// TIA Portal V17 program export: 0 tag tables, 0 data types, 33 data blocks, 57 code blocks (in call order from the OBs), 62 instance data blocks

DATA_BLOCK "DB_MainData"   // DB5001
{ S7_Optimized_Access := 'TRUE' }
VERSION : 0.1
// stored: AutoNumber false, DBAccessibleFromOPCUA true, DBAccessibleFromWebserver true, IsOnlyStoredInLoadMemory false, IsRetainMemResEnabled false, IsWriteProtectedInAS false, MemoryReserve 100
   VAR
      SafetyLevels { S7_SetPoint := 'True'} : "UDT_SafetyLevels";
      HMI { S7_SetPoint := 'True'} : "UDT_HMI";
      ManualModeActive : Bool := FALSE;
      MachineMode : UInt := 1;   // 0= No mode active, 1= Manual mode, 2= Homing mode, 3= Automatic mode
      AntennaEdge : Bool := FALSE;
      Antenna : Bool := FALSE;
   END_VAR
BEGIN
   SafetyLevels."Level_1L+" := FALSE;
   SafetyLevels."Level_2L+" := FALSE;
   SafetyLevels."Level_3L+" := TRUE;   // Doors + safety barriers + total stop
   SafetyLevels."Level_4L+" := FALSE;   // Doors + safety barriers + total stop + light barriers
   SafetyLevels."Level_5L+" := FALSE;   // Doors + safety barriers + total stop + turn table
   SafetyLevels."Level_6L+" := FALSE;
   SafetyLevels."Level_7L+" := FALSE;
   SafetyLevels."Level_8L+" := FALSE;
   SafetyLevels."Level_9L+" := FALSE;
   SafetyLevels."Level_10L+" := FALSE;
   SafetyLevels.SystemReady := TRUE;   // Doors + safety barriers + total stop + air pressure
   HMI.ScreenData[1] := 16#0001;
   HMI.ScreenData[2] := 16#0008;
   HMI.ScreenData[3] := 16#0000;
   HMI.ScreenData[4] := 16#0007;
   HMI.ScreenData[5] := 16#0000;
   HMI.UserNumber := 0;
   HMI.ActualScreenNumber := 8;
   HMI.RequiredScreenNumber := 0;
   HMI.FunctionKeys[1..8] := FALSE;
END_DATA_BLOCK

DATA_BLOCK "READER_DWELL"   // DB80
{ S7_Optimized_Access := 'TRUE' }
VERSION : 0.1
// stored: AutoNumber true, DBAccessibleFromOPCUA true, DBAccessibleFromWebserver true, IsOnlyStoredInLoadMemory false, IsRetainMemResEnabled false, IsWriteProtectedInAS false, MemoryReserve 100
   VAR
      DWELL_TMR : Array[0..16] of TON_TIME;
   END_VAR
BEGIN
END_DATA_BLOCK

DATA_BLOCK "Alarms"   // DB20
{ S7_Optimized_Access := 'FALSE' }
VERSION : 0.1
// stored: AutoNumber false, DBAccessibleFromOPCUA true, DBAccessibleFromWebserver true, IsOnlyStoredInLoadMemory false, IsWriteProtectedInAS false
   VAR
      Alarm : Array[1..256] of Bool;
      Warning : Array[1..256] of Bool;
      PartErrorsHMI : Array[1..256] of Bool;
      NOKInAuto : Bool := FALSE;
      Reset : Bool := FALSE;
      ResetHmi : Bool := FALSE;
      AlarmPLC : Array[0..100] of Bool;
   END_VAR
BEGIN
   Alarm[1..256] := FALSE;
   Warning[1..256] := FALSE;
   PartErrorsHMI[1..10] := FALSE;
   PartErrorsHMI[11] := TRUE;
   PartErrorsHMI[12..20] := FALSE;
   PartErrorsHMI[21] := TRUE;
   PartErrorsHMI[22..30] := FALSE;
   PartErrorsHMI[31] := TRUE;
   PartErrorsHMI[32..40] := FALSE;
   PartErrorsHMI[41] := TRUE;
   PartErrorsHMI[42..256] := FALSE;
   AlarmPLC[0..100] := FALSE;
END_DATA_BLOCK

DATA_BLOCK "AutoInfo"   // DB13
{ S7_Optimized_Access := 'TRUE' }
VERSION : 0.1
// stored: AutoNumber true, DBAccessibleFromOPCUA true, DBAccessibleFromWebserver true, IsOnlyStoredInLoadMemory false, IsRetainMemResEnabled false, IsWriteProtectedInAS false, MemoryReserve 100
   VAR
      EraseStation : Array[1..8] of Bool;
      ExtractedScan : String := '';
      EnableReferenceChange : Bool := TRUE;
   END_VAR
   VAR RETAIN
      R1BrakeTestRequired : Bool := TRUE;
      R1MasteringRequired : Bool := TRUE;
      PartMeasuredData { S7_SetPoint := 'True'} : "UDT_MeasuredPartData";
   END_VAR
   VAR
      EndProduction { S7_SetPoint := 'True'} : Bool;
   END_VAR
BEGIN
   EraseStation[1..8] := FALSE;
   PartMeasuredData.LeftCupforming.MaxForce := -7.98946;
   PartMeasuredData.LeftCupforming.MinimalWay := 9.841429;
   PartMeasuredData.LeftCupforming.MaxZposition := 55.44488;
   PartMeasuredData.LeftCupforming.OK := TRUE;
   PartMeasuredData.LeftCupforming.NOK := FALSE;
   PartMeasuredData.LeftCupforming.parameters.DigiforceProgram := 1;
   PartMeasuredData.LeftCupforming.parameters.FinalSpeed := 20.0;
   PartMeasuredData.LeftCupforming.parameters.ApproachSpeed := 100.0;
   PartMeasuredData.LeftCupforming.parameters.FinalForce := 80.0;
   PartMeasuredData.LeftCupforming.parameters.ApproachForce := 20.0;
   PartMeasuredData.LeftCupforming.parameters.EndWayImmediate := 9.9;
   PartMeasuredData.LeftCupforming.parameters.EndWayWithTimeout := 9.9;
   PartMeasuredData.LeftCupforming.parameters.SwitchingWay := 50.0;
   PartMeasuredData.LeftCupforming.parameters.EndWayTimeout := T#300MS;
   PartMeasuredData.RightCupforming.MaxForce := 8.163286;
   PartMeasuredData.RightCupforming.MinimalWay := 9.87697;
   PartMeasuredData.RightCupforming.MaxZposition := 56.52127;
   PartMeasuredData.RightCupforming.OK := TRUE;
   PartMeasuredData.RightCupforming.NOK := FALSE;
   PartMeasuredData.RightCupforming.parameters.DigiforceProgram := 1;
   PartMeasuredData.RightCupforming.parameters.FinalSpeed := 20.0;
   PartMeasuredData.RightCupforming.parameters.ApproachSpeed := 100.0;
   PartMeasuredData.RightCupforming.parameters.FinalForce := 80.0;
   PartMeasuredData.RightCupforming.parameters.ApproachForce := 20.0;
   PartMeasuredData.RightCupforming.parameters.EndWayImmediate := 9.9;
   PartMeasuredData.RightCupforming.parameters.EndWayWithTimeout := 9.9;
   PartMeasuredData.RightCupforming.parameters.SwitchingWay := 50.0;
   PartMeasuredData.RightCupforming.parameters.EndWayTimeout := T#300MS;
   PartMeasuredData.LeftRiveting1.Start := FALSE;
   PartMeasuredData.LeftRiveting1.PrgNumber := 0;
   PartMeasuredData.LeftRiveting1.Ready := FALSE;
   PartMeasuredData.LeftRiveting1.Running := FALSE;
   PartMeasuredData.LeftRiveting1.OK := FALSE;
   PartMeasuredData.LeftRiveting1.NOK := FALSE;
   PartMeasuredData.LeftRiveting1.H1OK := FALSE;
   PartMeasuredData.LeftRiveting1.H2OK := FALSE;
   PartMeasuredData.LeftRiveting1.TimeOK := FALSE;
   PartMeasuredData.LeftRiveting1.StartError := FALSE;
   PartMeasuredData.LeftRiveting1.LastH1 := 0.0;
   PartMeasuredData.LeftRiveting1.LastH2 := 0.0;
   PartMeasuredData.LeftRiveting1.LastTime := 0.0;
   PartMeasuredData.LeftRiveting1.LastZ1 := 0.0;
   PartMeasuredData.LeftRiveting1.Error := FALSE;
   PartMeasuredData.LeftRiveting1.NewData := FALSE;
   PartMeasuredData.LeftRiveting1.Z1OK := FALSE;
   PartMeasuredData.LeftRiveting1.NewDataAfterStart := FALSE;
   PartMeasuredData.LeftRiveting1.LastZ2 := 0.0;
   PartMeasuredData.LeftRiveting2.Start := FALSE;
   PartMeasuredData.LeftRiveting2.PrgNumber := 0;
   PartMeasuredData.LeftRiveting2.Ready := FALSE;
   PartMeasuredData.LeftRiveting2.Running := FALSE;
   PartMeasuredData.LeftRiveting2.OK := FALSE;
   PartMeasuredData.LeftRiveting2.NOK := FALSE;
   PartMeasuredData.LeftRiveting2.H1OK := FALSE;
   PartMeasuredData.LeftRiveting2.H2OK := FALSE;
   PartMeasuredData.LeftRiveting2.TimeOK := FALSE;
   PartMeasuredData.LeftRiveting2.StartError := FALSE;
   PartMeasuredData.LeftRiveting2.LastH1 := 0.0;
   PartMeasuredData.LeftRiveting2.LastH2 := 0.0;
   PartMeasuredData.LeftRiveting2.LastTime := 0.0;
   PartMeasuredData.LeftRiveting2.LastZ1 := 0.0;
   PartMeasuredData.LeftRiveting2.Error := FALSE;
   PartMeasuredData.LeftRiveting2.NewData := FALSE;
   PartMeasuredData.LeftRiveting2.Z1OK := FALSE;
   PartMeasuredData.LeftRiveting2.NewDataAfterStart := FALSE;
   PartMeasuredData.LeftRiveting2.LastZ2 := 0.0;
   PartMeasuredData.RightRiveting1.Start := FALSE;
   PartMeasuredData.RightRiveting1.PrgNumber := 0;
   PartMeasuredData.RightRiveting1.Ready := FALSE;
   PartMeasuredData.RightRiveting1.Running := FALSE;
   PartMeasuredData.RightRiveting1.OK := FALSE;
   PartMeasuredData.RightRiveting1.NOK := FALSE;
   PartMeasuredData.RightRiveting1.H1OK := FALSE;
   PartMeasuredData.RightRiveting1.H2OK := FALSE;
   PartMeasuredData.RightRiveting1.TimeOK := FALSE;
   PartMeasuredData.RightRiveting1.StartError := FALSE;
   PartMeasuredData.RightRiveting1.LastH1 := 0.0;
   PartMeasuredData.RightRiveting1.LastH2 := 0.0;
   PartMeasuredData.RightRiveting1.LastTime := 0.0;
   PartMeasuredData.RightRiveting1.LastZ1 := 0.0;
   PartMeasuredData.RightRiveting1.Error := FALSE;
   PartMeasuredData.RightRiveting1.NewData := FALSE;
   PartMeasuredData.RightRiveting1.Z1OK := FALSE;
   PartMeasuredData.RightRiveting1.NewDataAfterStart := FALSE;
   PartMeasuredData.RightRiveting1.LastZ2 := 0.0;
   PartMeasuredData.RightRiveting2.Start := FALSE;
   PartMeasuredData.RightRiveting2.PrgNumber := 0;
   PartMeasuredData.RightRiveting2.Ready := FALSE;
   PartMeasuredData.RightRiveting2.Running := FALSE;
   PartMeasuredData.RightRiveting2.OK := FALSE;
   PartMeasuredData.RightRiveting2.NOK := FALSE;
   PartMeasuredData.RightRiveting2.H1OK := FALSE;
   PartMeasuredData.RightRiveting2.H2OK := FALSE;
   PartMeasuredData.RightRiveting2.TimeOK := FALSE;
   PartMeasuredData.RightRiveting2.StartError := FALSE;
   PartMeasuredData.RightRiveting2.LastH1 := 0.0;
   PartMeasuredData.RightRiveting2.LastH2 := 0.0;
   PartMeasuredData.RightRiveting2.LastTime := 0.0;
   PartMeasuredData.RightRiveting2.LastZ1 := 0.0;
   PartMeasuredData.RightRiveting2.Error := FALSE;
   PartMeasuredData.RightRiveting2.NewData := FALSE;
   PartMeasuredData.RightRiveting2.Z1OK := FALSE;
   PartMeasuredData.RightRiveting2.NewDataAfterStart := FALSE;
   PartMeasuredData.RightRiveting2.LastZ2 := 0.0;
END_DATA_BLOCK

DATA_BLOCK "AutoPositions"   // DB11
{ S7_Optimized_Access := 'TRUE' }
VERSION : 0.1
// stored: AutoNumber true, DBAccessibleFromOPCUA true, DBAccessibleFromWebserver true, IsOnlyStoredInLoadMemory false, IsRetainMemResEnabled false, IsWriteProtectedInAS false, MemoryReserve 100
   VAR RETAIN
      St1_Table1 : "UDT_PositionData";
      St2_Table2 : "UDT_PositionData";
      St3_Fitting : "UDT_PositionData";
      R1_Gripper : "UDT_PositionData";
      AE_Gripper : "UDT_PositionData";
      St4_OKposition : "UDT_PositionData";
   END_VAR
   VAR
      emptyPos : "UDT_PositionData";
   END_VAR
BEGIN
END_DATA_BLOCK

DATA_BLOCK "St1Insertion"   // DB15
{ S7_Optimized_Access := 'TRUE' }
VERSION : 0.1
// stored: AutoNumber true, DBAccessibleFromOPCUA true, DBAccessibleFromWebserver true, IsOnlyStoredInLoadMemory false, IsRetainMemResEnabled false, IsWriteProtectedInAS false, MemoryReserve 100
   VAR
      ExpectedSensors : Array[0..20] of Bool;
      UsedSensors : Array[0..20] of Bool;
      SensorsState : Array[0..20] of Bool;
      SensorsNOK : Array[0..20] of Bool;
      NOKList : Array[0..20] of Int;
      InsertionOK : Bool := TRUE;
      InsertionNOK : Bool := FALSE;
      InsertionEmpty : Bool := TRUE;
      EmptyBits : Array[0..20] of Bool;
      FullBits : Array[0..20] of Bool;
   END_VAR
BEGIN
   ExpectedSensors[0..20] := FALSE;
   UsedSensors[0..20] := FALSE;
   SensorsState[0..20] := FALSE;
   SensorsNOK[0..20] := FALSE;
   NOKList[0..20] := 0;
   EmptyBits[0..20] := FALSE;
   FullBits[0] := FALSE;
   FullBits[1..17] := TRUE;
   FullBits[18..20] := FALSE;
END_DATA_BLOCK

DATA_BLOCK "CylindersDowngrade"   // DB37
{ S7_Optimized_Access := 'TRUE' }
VERSION : 0.1
// stored: AutoNumber true, DBAccessibleFromOPCUA true, DBAccessibleFromWebserver true, IsOnlyStoredInLoadMemory false, IsRetainMemResEnabled false, IsWriteProtectedInAS false, MemoryReserve 100
   VAR RETAIN
      V302UseAnalogForBP : Bool := FALSE;
   END_VAR
BEGIN
END_DATA_BLOCK

DATA_BLOCK "Cylinders_Commands"   // DB12
{ S7_Optimized_Access := 'FALSE' }
VERSION : 0.1
// stored: AutoNumber false, DBAccessibleFromOPCUA true, DBAccessibleFromWebserver true, IsOnlyStoredInLoadMemory false, IsWriteProtectedInAS false
   VAR RETAIN
      VH1 { S7_SetPoint := 'True'} : "UDT_HydraulicCylinderData";
      VH2 { S7_SetPoint := 'True'} : "UDT_HydraulicCylinderData";
      VH3 { S7_SetPoint := 'True'} : "UDT_HydraulicCylinderData";
      VH4 { S7_SetPoint := 'True'} : "UDT_HydraulicCylinderData";
   END_VAR
BEGIN
   VH1.Pressure := 0.0;
   VH1.Flow := 0.0;
   VH1.Position := 0.0;
   VH1.StandstillPosition := 0.0;
   VH1.PressureCmd := 0.0;
   VH1.FlowCmd := 0.0;
   VH1.PressureBack := 0.0;
   VH1.FlowBack := 0.0;
   VH1.HAxis := 0.0;
   VH1.Force := 0.0;
   VH1.Status.InWp := FALSE;
   VH1.Status.InBp := FALSE;
   VH1.Status.InFp := FALSE;
   VH1.Status.ToWp := FALSE;
   VH1.Status.ToBp := FALSE;
   VH1.Status.ToFp := FALSE;
   VH1.InBp_1mm_margin := FALSE;
   VH2.Pressure := 0.0;
   VH2.Flow := 0.0;
   VH2.Position := 0.0;
   VH2.StandstillPosition := 0.0;
   VH2.PressureCmd := 0.0;
   VH2.FlowCmd := 0.0;
   VH2.PressureBack := 0.0;
   VH2.FlowBack := 0.0;
   VH2.HAxis := 0.0;
   VH2.Force := 0.0;
   VH2.Status.InWp := FALSE;
   VH2.Status.InBp := FALSE;
   VH2.Status.InFp := FALSE;
   VH2.Status.ToWp := FALSE;
   VH2.Status.ToBp := FALSE;
   VH2.Status.ToFp := FALSE;
   VH2.InBp_1mm_margin := FALSE;
   VH3.Pressure := 0.0;
   VH3.Flow := 0.0;
   VH3.Position := 5.820313;
   VH3.StandstillPosition := 0.0;
   VH3.PressureCmd := 0.0;
   VH3.FlowCmd := 0.0;
   VH3.PressureBack := 0.0;
   VH3.FlowBack := 0.0;
   VH3.HAxis := 0.0;
   VH3.Force := 0.0;
   VH3.Status.InWp := FALSE;
   VH3.Status.InBp := FALSE;
   VH3.Status.InFp := FALSE;
   VH3.Status.ToWp := FALSE;
   VH3.Status.ToBp := FALSE;
   VH3.Status.ToFp := FALSE;
   VH3.InBp_1mm_margin := FALSE;
   VH4.Pressure := 0.0;
   VH4.Flow := 0.0;
   VH4.Position := 4.661458;
   VH4.StandstillPosition := 0.0;
   VH4.PressureCmd := 0.0;
   VH4.FlowCmd := 0.0;
   VH4.PressureBack := 0.0;
   VH4.FlowBack := 0.0;
   VH4.HAxis := 0.0;
   VH4.Force := 0.0;
   VH4.Status.InWp := FALSE;
   VH4.Status.InBp := FALSE;
   VH4.Status.InFp := FALSE;
   VH4.Status.ToWp := FALSE;
   VH4.Status.ToBp := FALSE;
   VH4.Status.ToFp := FALSE;
   VH4.InBp_1mm_margin := FALSE;
END_DATA_BLOCK

DATA_BLOCK "DevicesData"   // DB26
{ S7_Optimized_Access := 'FALSE' }
VERSION : 0.1
// stored: AutoNumber false, DBAccessibleFromOPCUA true, DBAccessibleFromWebserver true, IsOnlyStoredInLoadMemory false, IsWriteProtectedInAS false
   VAR
      scanner { S7_SetPoint := 'True'} : "UDT_Reader";
      TurnTable { S7_SetPoint := 'True'} : "UDT_TurnTable";
      rivetingLeft_cycle { S7_SetPoint := 'True'} : "UDT_FittingStatus";
      rivetingRight_cycle { S7_SetPoint := 'True'} : "UDT_FittingStatus";
      cupformingLeft_cycle { S7_SetPoint := 'True'} : "UDT_FittingStatus";
      cupformingRight_cycle { S7_SetPoint := 'True'} : "UDT_FittingStatus";
      R1 { S7_SetPoint := 'True'} : "UDT_Robot";
      R2 { S7_SetPoint := 'True'} : "UDT_Robot";
      Digiforce1 { S7_SetPoint := 'True'} : "UDT_Digiforce";
      Digiforce2 { S7_SetPoint := 'True'} : "UDT_Digiforce";
      Cylinders : Array[0.."NumberOfCylinders"] of "UDT_Cylinder";
      cupformingLeft_cylinder { S7_SetPoint := 'True'} : "UDT_HydraulicCylinderData";
      cupformingRight_cylinder { S7_SetPoint := 'True'} : "UDT_HydraulicCylinderData";
      CupformingPressure : Real := 80.0;
      Hydraulic { S7_SetPoint := 'True'} : "UDT_HydraulicPump";
      "TA1-3MA" { S7_SetPoint := 'True'} : "UDT_Servo";
      Friedrich1 { S7_SetPoint := 'True'} : "UDT_Friedrich";
      Friedrich2 { S7_SetPoint := 'True'} : "UDT_Friedrich";
      Camera : Array[1..4] of "UDT_Camera_Keyence_IV";
   END_VAR
BEGIN
   scanner.start := FALSE;
   scanner.ready := FALSE;
   scanner.error := FALSE;
   scanner.newData := FALSE;
   scanner.bankNr := 0;
   scanner.errorID := 16#0000;
   scanner.length := 6;
   scanner.data := 'NoRead';
   TurnTable.Commands.ManualMode.ReadyToJogCW := FALSE;
   TurnTable.Commands.ManualMode.JogCW := FALSE;
   TurnTable.Commands.ManualMode.ReadyToJogCCW := FALSE;
   TurnTable.Commands.ManualMode.JogCCW := FALSE;
   TurnTable.Commands.ManualMode.ReadyToStartCW := FALSE;
   TurnTable.Commands.ManualMode.StartCW := FALSE;
   TurnTable.Commands.ManualMode.ReadyToStartCCW := FALSE;
   TurnTable.Commands.ManualMode.StartCCW := FALSE;
   TurnTable.Commands.AutomaticMode.ReadyToJogCW := FALSE;
   TurnTable.Commands.AutomaticMode.JogCW := FALSE;
   TurnTable.Commands.AutomaticMode.ReadyToJogCCW := FALSE;
   TurnTable.Commands.AutomaticMode.JogCCW := FALSE;
   TurnTable.Commands.AutomaticMode.ReadyToStartCW := FALSE;
   TurnTable.Commands.AutomaticMode.StartCW := FALSE;
   TurnTable.Commands.AutomaticMode.ReadyToStartCCW := FALSE;
   TurnTable.Commands.AutomaticMode.StartCCW := FALSE;
   TurnTable.Status.Collision := FALSE;
   TurnTable.Status.Communication := FALSE;
   TurnTable.Status.EnabledForOneScan := FALSE;
   TurnTable.Status.IndexerInPositionForOneScan := FALSE;
   TurnTable.Status.CycleStep := 0;
   TurnTable.Status.CycleRunning := FALSE;
   TurnTable.Status.CycleFinished := TRUE;
   TurnTable.Status.CycleStopped := FALSE;
   TurnTable.Status.DoneCW := FALSE;
   TurnTable.Status.DoneCCW := FALSE;
   TurnTable.Status.SafetyPosition := TRUE;
   TurnTable.Status.BasicPosition := TRUE;
   TurnTable."I/O".iTurnTableInSafetyPosition := TRUE;
   TurnTable."I/O".Inputs.ReadyToEnable := TRUE;
   TurnTable."I/O".Inputs.EnableActive := TRUE;
   TurnTable."I/O".Inputs.Enabled := TRUE;
   TurnTable."I/O".Inputs.ReadyToStart := TRUE;
   TurnTable."I/O".Inputs.Operating := FALSE;
   TurnTable."I/O".Inputs.IndexerInPosition := TRUE;
   TurnTable."I/O".Inputs.StopIsSelected := FALSE;
   TurnTable."I/O".Inputs.AlarmTimeout := FALSE;
   TurnTable."I/O".Inputs.AlarmPositionRunOver := FALSE;
   TurnTable."I/O".Inputs.AlarmSafety := FALSE;
   TurnTable."I/O".Inputs.SumError := FALSE;
   TurnTable."I/O".Inputs.SumWarning := FALSE;
   TurnTable."I/O".Inputs.STOIsSelected := FALSE;
   TurnTable."I/O".Inputs.STOIsActive := FALSE;
   TurnTable."I/O".Inputs.WatchdogSend := TRUE;
   TurnTable."I/O".Outputs.Enable := FALSE;
   TurnTable."I/O".Outputs.Stop := FALSE;
   TurnTable."I/O".Outputs.CycleCW := FALSE;
   TurnTable."I/O".Outputs.CycleCCW := FALSE;
   TurnTable."I/O".Outputs.JogCW := FALSE;
   TurnTable."I/O".Outputs.JogCCW := FALSE;
   TurnTable."I/O".Outputs.ResetError := FALSE;
   TurnTable."I/O".Outputs.WatchdogReceive := FALSE;
   cupformingLeft_cycle.Start := FALSE;
   cupformingLeft_cycle.Done := FALSE;
   cupformingLeft_cycle.Running := FALSE;
   cupformingLeft_cycle.Returning := FALSE;
   cupformingLeft_cycle.OK := TRUE;
   cupformingLeft_cycle.ContinueFitting := TRUE;
   cupformingLeft_cycle.ContinueReturn := TRUE;
   cupformingLeft_cycle.InPreposition := FALSE;
   cupformingLeft_cycle.continueWithSupportToWork := TRUE;
   cupformingLeft_cycle.StartSequence := FALSE;
   cupformingLeft_cycle.DoneSequence := FALSE;
   cupformingLeft_cycle.PartErrors[1..8] := FALSE;
   cupformingLeft_cycle.rivetStatus := 0;
   cupformingRight_cycle.Start := FALSE;
   cupformingRight_cycle.Done := FALSE;
   cupformingRight_cycle.Running := FALSE;
   cupformingRight_cycle.Returning := FALSE;
   cupformingRight_cycle.OK := TRUE;
   cupformingRight_cycle.ContinueFitting := TRUE;
   cupformingRight_cycle.ContinueReturn := TRUE;
   cupformingRight_cycle.InPreposition := FALSE;
   cupformingRight_cycle.continueWithSupportToWork := TRUE;
   cupformingRight_cycle.StartSequence := FALSE;
   cupformingRight_cycle.DoneSequence := FALSE;
   cupformingRight_cycle.PartErrors[1..8] := FALSE;
   cupformingRight_cycle.rivetStatus := 0;
   R1.StartReq := FALSE;
   R1.StartAllowed := FALSE;
   R1.Started := FALSE;
   R1.Job.JobNr := 16#05;
   R1.Job.Start := FALSE;
   R1.Job.Done := FALSE;
   R2.StartReq := FALSE;
   R2.StartAllowed := FALSE;
   R2.Started := FALSE;
   R2.Job.JobNr := 16#00;
   R2.Job.Start := FALSE;
   R2.Job.Done := FALSE;
   Digiforce1.programActual := 0;
   Digiforce1.programOK := TRUE;
   Digiforce1.ProgramChangeNOK := FALSE;
   Digiforce1.programSet := 0;
   Digiforce1.ActualWay := 8.027563;
   Digiforce1.ActualForce := 0.0;
   Digiforce1.Ready := TRUE;
   Digiforce1.ResultOK := TRUE;
   Digiforce1.ResultNOK := FALSE;
   Digiforce1.Auto := FALSE;
   Digiforce1.Start := FALSE;
   Digiforce1.Running := FALSE;
   Digiforce1.TareX := FALSE;
   Digiforce2.programActual := 0;
   Digiforce2.programOK := TRUE;
   Digiforce2.ProgramChangeNOK := FALSE;
   Digiforce2.programSet := 0;
   Digiforce2.ActualWay := 8.029956;
   Digiforce2.ActualForce := 0.0;
   Digiforce2.Ready := TRUE;
   Digiforce2.ResultOK := TRUE;
   Digiforce2.ResultNOK := FALSE;
   Digiforce2.Auto := FALSE;
   Digiforce2.Start := FALSE;
   Digiforce2.Running := FALSE;
   Digiforce2.TareX := FALSE;
   Cylinders[0..6].InWp := FALSE;
   Cylinders[7..8].InWp := TRUE;
   Cylinders[9..16].InWp := FALSE;
   Cylinders[17..18].InWp := TRUE;
   Cylinders[19].InWp := FALSE;
   Cylinders[0..6].InBp := TRUE;
   Cylinders[7..8].InBp := FALSE;
   Cylinders[9..16].InBp := TRUE;
   Cylinders[17..19].InBp := FALSE;
   Cylinders[0..4].InFp := FALSE;
   Cylinders[5..6].InFp := TRUE;
   Cylinders[7..8].InFp := FALSE;
   Cylinders[9..18].InFp := TRUE;
   Cylinders[19].InFp := FALSE;
   Cylinders[0..6].ToWp := FALSE;
   Cylinders[7..8].ToWp := TRUE;
   Cylinders[9..19].ToWp := FALSE;
   Cylinders[0..4].ToBp := TRUE;
   Cylinders[5..19].ToBp := FALSE;
   Cylinders[0..4].ToFp := FALSE;
   Cylinders[5..6].ToFp := TRUE;
   Cylinders[7..8].ToFp := FALSE;
   Cylinders[9..18].ToFp := TRUE;
   Cylinders[19].ToFp := FALSE;
   cupformingLeft_cylinder.Pressure := 0.0;
   cupformingLeft_cylinder.Flow := 0.0;
   cupformingLeft_cylinder.Position := 0.1801215;
   cupformingLeft_cylinder.StandstillPosition := 0.1974826;
   cupformingLeft_cylinder.PressureCmd := 80.0;
   cupformingLeft_cylinder.FlowCmd := 100.0;
   cupformingLeft_cylinder.PressureBack := 0.0;
   cupformingLeft_cylinder.FlowBack := 0.0;
   cupformingLeft_cylinder.HAxis := 8.058673;
   cupformingLeft_cylinder.Force := 0.2526712;
   cupformingLeft_cylinder.Status.InWp := FALSE;
   cupformingLeft_cylinder.Status.InBp := TRUE;
   cupformingLeft_cylinder.Status.InFp := TRUE;
   cupformingLeft_cylinder.Status.ToWp := FALSE;
   cupformingLeft_cylinder.Status.ToBp := FALSE;
   cupformingLeft_cylinder.Status.ToFp := TRUE;
   cupformingLeft_cylinder.InBp_1mm_margin := FALSE;
   cupformingRight_cylinder.Pressure := 0.0;
   cupformingRight_cylinder.Flow := 0.0;
   cupformingRight_cylinder.Position := 0.249566;
   cupformingRight_cylinder.StandstillPosition := 0.2625868;
   cupformingRight_cylinder.PressureCmd := 80.0;
   cupformingRight_cylinder.FlowCmd := 100.0;
   cupformingRight_cylinder.PressureBack := 0.0;
   cupformingRight_cylinder.FlowBack := 0.0;
   cupformingRight_cylinder.HAxis := 8.017026;
   cupformingRight_cylinder.Force := -0.1702255;
   cupformingRight_cylinder.Status.InWp := FALSE;
   cupformingRight_cylinder.Status.InBp := TRUE;
   cupformingRight_cylinder.Status.InFp := TRUE;
   cupformingRight_cylinder.Status.ToWp := FALSE;
   cupformingRight_cylinder.Status.ToBp := FALSE;
   cupformingRight_cylinder.Status.ToFp := TRUE;
   cupformingRight_cylinder.InBp_1mm_margin := FALSE;
   Hydraulic.OilLevel := 0.0;
   Hydraulic.OilTemperature := 0.0;
   Hydraulic.OilPressure := 0.0;
   Hydraulic.AutoMode := FALSE;
   Hydraulic.TemperatureError := FALSE;
   Hydraulic.LevelError := FALSE;
   Hydraulic.PressureError := FALSE;
   Hydraulic.AutoModeReady := FALSE;
END_DATA_BLOCK

DATA_BLOCK "DB_EksData"   // DB5052
{ S7_Optimized_Access := 'TRUE' }
VERSION : 0.1
// stored: AutoNumber false, DBAccessibleFromOPCUA true, DBAccessibleFromWebserver true, IsOnlyStoredInLoadMemory false, IsRetainMemResEnabled false, IsWriteProtectedInAS false, MemoryReserve 0
   VAR
      EmptyKey { S7_SetPoint := 'True'} : "UDT_EksKey";
      LoadedData { S7_SetPoint := 'True'} : "UDT_EksKey";
      ActualKey { S7_SetPoint := 'True'} : "UDT_EksKey";
      LastKey { S7_SetPoint := 'True'} : "UDT_EksKey";
      KeyListHMI { S7_SetPoint := 'True'} : Array[1..10] of "UDT_EksKey";
   END_VAR
BEGIN
   EmptyKey.Level := 0;
   EmptyKey.EmployeeID[1..4] := ' ';
   EmptyKey.KeyID[1..16] := ' ';
   EmptyKey.Comment[1..20] := ' ';
   LoadedData.Level := 0;
   LoadedData.EmployeeID[1..4] := ' ';
   LoadedData.KeyID[1] := '0';
   LoadedData.KeyID[2] := '3';
   LoadedData.KeyID[3] := '7';
   LoadedData.KeyID[4] := '2';
   LoadedData.KeyID[5] := '4';
   LoadedData.KeyID[6] := '5';
   LoadedData.KeyID[7] := '2';
   LoadedData.KeyID[8] := '9';
   LoadedData.KeyID[9] := 'A';
   LoadedData.KeyID[10] := '6';
   LoadedData.KeyID[11..12] := '0';
   LoadedData.KeyID[13] := '1';
   LoadedData.KeyID[14] := '0';
   LoadedData.KeyID[15] := '3';
   LoadedData.KeyID[16] := '2';
   LoadedData.Comment[1..20] := ' ';
   ActualKey.Level := 5;
   ActualKey.EmployeeID[1..4] := ' ';
   ActualKey.KeyID[1] := '0';
   ActualKey.KeyID[2] := '3';
   ActualKey.KeyID[3] := '7';
   ActualKey.KeyID[4] := '2';
   ActualKey.KeyID[5] := '4';
   ActualKey.KeyID[6] := '5';
   ActualKey.KeyID[7] := '2';
   ActualKey.KeyID[8] := '9';
   ActualKey.KeyID[9] := 'A';
   ActualKey.KeyID[10] := '6';
   ActualKey.KeyID[11..12] := '0';
   ActualKey.KeyID[13] := '1';
   ActualKey.KeyID[14] := '0';
   ActualKey.KeyID[15] := '3';
   ActualKey.KeyID[16] := '2';
   ActualKey.Comment[1..20] := ' ';
   LastKey.Level := 0;
   LastKey.EmployeeID[1..4] := ' ';
   LastKey.KeyID[1..16] := ' ';
   LastKey.Comment[1..20] := ' ';
   KeyListHMI[1..10].Level := 0;
   KeyListHMI[1].EmployeeID[1..4] := ' ';
   KeyListHMI[2].EmployeeID[1..4] := ' ';
   KeyListHMI[3].EmployeeID[1..4] := ' ';
   KeyListHMI[4].EmployeeID[1..4] := ' ';
   KeyListHMI[5].EmployeeID[1..4] := ' ';
   KeyListHMI[6].EmployeeID[1..4] := ' ';
   KeyListHMI[7].EmployeeID[1..4] := ' ';
   KeyListHMI[8].EmployeeID[1..4] := ' ';
   KeyListHMI[9].EmployeeID[1..4] := ' ';
   KeyListHMI[10].EmployeeID[1..4] := ' ';
   KeyListHMI[1].KeyID[1..16] := ' ';
   KeyListHMI[2].KeyID[1..16] := ' ';
   KeyListHMI[3].KeyID[1..16] := ' ';
   KeyListHMI[4].KeyID[1..16] := ' ';
   KeyListHMI[5].KeyID[1..16] := ' ';
   KeyListHMI[6].KeyID[1..16] := ' ';
   KeyListHMI[7].KeyID[1..16] := ' ';
   KeyListHMI[8].KeyID[1..16] := ' ';
   KeyListHMI[9].KeyID[1..16] := ' ';
   KeyListHMI[10].KeyID[1..16] := ' ';
   KeyListHMI[1].Comment[1..20] := ' ';
   KeyListHMI[2].Comment[1..20] := ' ';
   KeyListHMI[3].Comment[1..20] := ' ';
   KeyListHMI[4].Comment[1..20] := ' ';
   KeyListHMI[5].Comment[1..20] := ' ';
   KeyListHMI[6].Comment[1..20] := ' ';
   KeyListHMI[7].Comment[1..20] := ' ';
   KeyListHMI[8].Comment[1..20] := ' ';
   KeyListHMI[9].Comment[1..20] := ' ';
   KeyListHMI[10].Comment[1..20] := ' ';
END_DATA_BLOCK

DATA_BLOCK "DB_EksList"   // DB5051
{ S7_Optimized_Access := 'TRUE' }
VERSION : 0.1
// stored: AutoNumber false, DBAccessibleFromOPCUA true, DBAccessibleFromWebserver true, IsOnlyStoredInLoadMemory false, IsRetainMemResEnabled false, IsWriteProtectedInAS false, MemoryReserve 100
   VAR RETAIN
      Key { S7_SetPoint := 'True'} : Array[1.."EksNumberOfKeys"] of "UDT_EksKey";
   END_VAR
BEGIN
   Key[1..5].Level := 5;
   Key[6..9].Level := 3;
   Key[10..13].Level := 2;
   Key[14..18].Level := 5;
   Key[19..100].Level := 0;
   Key[1].EmployeeID[1..4] := ' ';
   Key[2].EmployeeID[1] := '¥';
   Key[2].EmployeeID[2] := 'Z';
   Key[2].EmployeeID[3] := '¥';
   Key[2].EmployeeID[4] := 'Z';
   Key[3].EmployeeID[1..4] := ' ';
   Key[4].EmployeeID[1..4] := ' ';
   Key[5].EmployeeID[1..4] := ' ';
   Key[6].EmployeeID[1..4] := ' ';
   Key[7].EmployeeID[1..4] := ' ';
   Key[8].EmployeeID[1..4] := ' ';
   Key[9].EmployeeID[1..4] := ' ';
   Key[10].EmployeeID[1..4] := ' ';
   Key[11].EmployeeID[1..4] := ' ';
   Key[12].EmployeeID[1..4] := ' ';
   Key[13].EmployeeID[1..4] := ' ';
   Key[14].EmployeeID[1..4] := ' ';
   Key[15].EmployeeID[1..4] := ' ';
   Key[16].EmployeeID[1..4] := ' ';
   Key[17].EmployeeID[1..4] := ' ';
   Key[18].EmployeeID[1..4] := ' ';
   Key[19].EmployeeID[1..4] := ' ';
   Key[20].EmployeeID[1..4] := ' ';
   Key[21].EmployeeID[1..4] := ' ';
   Key[22].EmployeeID[1..4] := ' ';
   Key[23].EmployeeID[1..4] := ' ';
   Key[24].EmployeeID[1..4] := ' ';
   Key[25].EmployeeID[1..4] := ' ';
   Key[26].EmployeeID[1..4] := ' ';
   Key[27].EmployeeID[1..4] := ' ';
   Key[28].EmployeeID[1..4] := ' ';
   Key[29].EmployeeID[1..4] := ' ';
   Key[30].EmployeeID[1..4] := ' ';
   Key[31].EmployeeID[1..4] := ' ';
   Key[32].EmployeeID[1..4] := ' ';
   Key[33].EmployeeID[1..4] := ' ';
   Key[34].EmployeeID[1..4] := ' ';
   Key[35].EmployeeID[1..4] := ' ';
   Key[36].EmployeeID[1..4] := ' ';
   Key[37].EmployeeID[1..4] := ' ';
   Key[38].EmployeeID[1..4] := ' ';
   Key[39].EmployeeID[1..4] := ' ';
   Key[40].EmployeeID[1..4] := ' ';
   Key[41].EmployeeID[1..4] := ' ';
   Key[42].EmployeeID[1..4] := ' ';
   Key[43].EmployeeID[1..4] := ' ';
   Key[44].EmployeeID[1..4] := ' ';
   Key[45].EmployeeID[1..4] := ' ';
   Key[46].EmployeeID[1..4] := ' ';
   Key[47].EmployeeID[1..4] := ' ';
   Key[48].EmployeeID[1..4] := ' ';
   Key[49].EmployeeID[1..4] := ' ';
   Key[50].EmployeeID[1..4] := ' ';
   Key[51].EmployeeID[1..4] := ' ';
   Key[52].EmployeeID[1..4] := ' ';
   Key[53].EmployeeID[1..4] := ' ';
   Key[54].EmployeeID[1..4] := ' ';
   Key[55].EmployeeID[1..4] := ' ';
   Key[56].EmployeeID[1..4] := ' ';
   Key[57].EmployeeID[1..4] := ' ';
   Key[58].EmployeeID[1..4] := ' ';
   Key[59].EmployeeID[1..4] := ' ';
   Key[60].EmployeeID[1..4] := ' ';
   Key[61].EmployeeID[1..4] := ' ';
   Key[62].EmployeeID[1..4] := ' ';
   Key[63].EmployeeID[1..4] := ' ';
   Key[64].EmployeeID[1..4] := ' ';
   Key[65].EmployeeID[1..4] := ' ';
   Key[66].EmployeeID[1..4] := ' ';
   Key[67].EmployeeID[1..4] := ' ';
   Key[68].EmployeeID[1..4] := ' ';
   Key[69].EmployeeID[1..4] := ' ';
   Key[70].EmployeeID[1..4] := ' ';
   Key[71].EmployeeID[1..4] := ' ';
   Key[72].EmployeeID[1..4] := ' ';
   Key[73].EmployeeID[1..4] := ' ';
   Key[74].EmployeeID[1..4] := ' ';
   Key[75].EmployeeID[1..4] := ' ';
   Key[76].EmployeeID[1..4] := ' ';
   Key[77].EmployeeID[1..4] := ' ';
   Key[78].EmployeeID[1..4] := ' ';
   Key[79].EmployeeID[1..4] := ' ';
   Key[80].EmployeeID[1..4] := ' ';
   Key[81].EmployeeID[1..4] := ' ';
   Key[82].EmployeeID[1..4] := ' ';
   Key[83].EmployeeID[1..4] := ' ';
   Key[84].EmployeeID[1..4] := ' ';
   Key[85].EmployeeID[1..4] := ' ';
   Key[86].EmployeeID[1..4] := ' ';
   Key[87].EmployeeID[1..4] := ' ';
   Key[88].EmployeeID[1..4] := ' ';
   Key[89].EmployeeID[1..4] := ' ';
   Key[90].EmployeeID[1..4] := ' ';
   Key[91].EmployeeID[1..4] := ' ';
   Key[92].EmployeeID[1..4] := ' ';
   Key[93].EmployeeID[1..4] := ' ';
   Key[94].EmployeeID[1..4] := ' ';
   Key[95].EmployeeID[1..4] := ' ';
   Key[96].EmployeeID[1..4] := ' ';
   Key[97].EmployeeID[1..4] := ' ';
   Key[98].EmployeeID[1..4] := ' ';
   Key[99].EmployeeID[1..4] := ' ';
   Key[100].EmployeeID[1..4] := ' ';
   Key[1].KeyID[1] := '0';
   Key[1].KeyID[2] := '3';
   Key[1].KeyID[3] := '6';
   Key[1].KeyID[4] := 'C';
   Key[1].KeyID[5] := 'B';
   Key[1].KeyID[6] := 'C';
   Key[1].KeyID[7] := 'F';
   Key[1].KeyID[8] := '4';
   Key[1].KeyID[9] := '0';
   Key[1].KeyID[10] := 'F';
   Key[1].KeyID[11..12] := '0';
   Key[1].KeyID[13] := '1';
   Key[1].KeyID[14] := '0';
   Key[1].KeyID[15] := '3';
   Key[1].KeyID[16] := '2';
   Key[2].KeyID[1] := '0';
   Key[2].KeyID[2..3] := '3';
   Key[2].KeyID[4] := 'E';
   Key[2].KeyID[5] := '0';
   Key[2].KeyID[6] := '2';
   Key[2].KeyID[7] := 'E';
   Key[2].KeyID[8] := '5';
   Key[2].KeyID[9] := 'C';
   Key[2].KeyID[10] := 'B';
   Key[2].KeyID[11..12] := '0';
   Key[2].KeyID[13] := '1';
   Key[2].KeyID[14] := '0';
   Key[2].KeyID[15] := '3';
   Key[2].KeyID[16] := '2';
   Key[3].KeyID[1] := '0';
   Key[3].KeyID[2] := '3';
   Key[3].KeyID[3] := '7';
   Key[3].KeyID[4] := '2';
   Key[3].KeyID[5] := '4';
   Key[3].KeyID[6] := '5';
   Key[3].KeyID[7] := '2';
   Key[3].KeyID[8] := '9';
   Key[3].KeyID[9] := 'A';
   Key[3].KeyID[10] := '6';
   Key[3].KeyID[11..12] := '0';
   Key[3].KeyID[13] := '1';
   Key[3].KeyID[14] := '0';
   Key[3].KeyID[15] := '3';
   Key[3].KeyID[16] := '2';
   Key[4].KeyID[1] := '0';
   Key[4].KeyID[2] := '3';
   Key[4].KeyID[3] := '7';
   Key[4].KeyID[4] := '2';
   Key[4].KeyID[5..6] := '5';
   Key[4].KeyID[7] := '9';
   Key[4].KeyID[8] := 'D';
   Key[4].KeyID[9] := '8';
   Key[4].KeyID[10] := 'A';
   Key[4].KeyID[11..12] := '0';
   Key[4].KeyID[13] := '1';
   Key[4].KeyID[14] := '0';
   Key[4].KeyID[15] := '3';
   Key[4].KeyID[16] := '2';
   Key[5].KeyID[1] := '0';
   Key[5].KeyID[2] := '3';
   Key[5].KeyID[3] := '7';
   Key[5].KeyID[4] := '2';
   Key[5].KeyID[5] := '4';
   Key[5].KeyID[6] := '3';
   Key[5].KeyID[7] := 'B';
   Key[5].KeyID[8] := 'A';
   Key[5].KeyID[9] := '3';
   Key[5].KeyID[10] := 'F';
   Key[5].KeyID[11..12] := '0';
   Key[5].KeyID[13] := '1';
   Key[5].KeyID[14] := '0';
   Key[5].KeyID[15] := '3';
   Key[5].KeyID[16] := '2';
   Key[6].KeyID[1] := '0';
   Key[6].KeyID[2] := '3';
   Key[6].KeyID[3] := '7';
   Key[6].KeyID[4] := '2';
   Key[6].KeyID[5] := '9';
   Key[6].KeyID[6] := '7';
   Key[6].KeyID[7] := '0';
   Key[6].KeyID[8] := 'C';
   Key[6].KeyID[9] := '2';
   Key[6].KeyID[10] := 'A';
   Key[6].KeyID[11..12] := '0';
   Key[6].KeyID[13] := '1';
   Key[6].KeyID[14] := '0';
   Key[6].KeyID[15] := '3';
   Key[6].KeyID[16] := '2';
   Key[7].KeyID[1] := '0';
   Key[7].KeyID[2] := '3';
   Key[7].KeyID[3] := '7';
   Key[7].KeyID[4] := '3';
   Key[7].KeyID[5] := '0';
   Key[7].KeyID[6] := 'A';
   Key[7].KeyID[7] := 'D';
   Key[7].KeyID[8] := '7';
   Key[7].KeyID[9] := '0';
   Key[7].KeyID[10] := '1';
   Key[7].KeyID[11..12] := '0';
   Key[7].KeyID[13] := '1';
   Key[7].KeyID[14] := '0';
   Key[7].KeyID[15] := '3';
   Key[7].KeyID[16] := '2';
   Key[8].KeyID[1] := '0';
   Key[8].KeyID[2] := '3';
   Key[8].KeyID[3] := '7';
   Key[8].KeyID[4] := '2';
   Key[8].KeyID[5] := '4';
   Key[8].KeyID[6..7] := '5';
   Key[8].KeyID[8..9] := 'F';
   Key[8].KeyID[10] := 'B';
   Key[8].KeyID[11..12] := '0';
   Key[8].KeyID[13] := '1';
   Key[8].KeyID[14] := '0';
   Key[8].KeyID[15] := '3';
   Key[8].KeyID[16] := '2';
   Key[9].KeyID[1] := '0';
   Key[9].KeyID[2] := '3';
   Key[9].KeyID[3] := '7';
   Key[9].KeyID[4] := '2';
   Key[9].KeyID[5] := '9';
   Key[9].KeyID[6] := 'C';
   Key[9].KeyID[7] := '3';
   Key[9].KeyID[8] := '8';
   Key[9].KeyID[9] := '3';
   Key[9].KeyID[10] := '2';
   Key[9].KeyID[11..12] := '0';
   Key[9].KeyID[13] := '1';
   Key[9].KeyID[14] := '0';
   Key[9].KeyID[15] := '3';
   Key[9].KeyID[16] := '2';
   Key[10].KeyID[1] := '0';
   Key[10].KeyID[2] := '3';
   Key[10].KeyID[3] := '7';
   Key[10].KeyID[4] := '2';
   Key[10].KeyID[5] := 'C';
   Key[10].KeyID[6..7] := '3';
   Key[10].KeyID[8] := 'E';
   Key[10].KeyID[9] := 'B';
   Key[10].KeyID[10] := '6';
   Key[10].KeyID[11..12] := '0';
   Key[10].KeyID[13] := '1';
   Key[10].KeyID[14] := '0';
   Key[10].KeyID[15] := '3';
   Key[10].KeyID[16] := '2';
   Key[11].KeyID[1] := '0';
   Key[11].KeyID[2] := '3';
   Key[11].KeyID[3] := '7';
   Key[11].KeyID[4] := '3';
   Key[11].KeyID[5] := '0';
   Key[11].KeyID[6] := 'C';
   Key[11].KeyID[7] := '3';
   Key[11].KeyID[8] := '0';
   Key[11].KeyID[9] := 'B';
   Key[11].KeyID[10] := 'F';
   Key[11].KeyID[11..12] := '0';
   Key[11].KeyID[13] := '1';
   Key[11].KeyID[14] := '0';
   Key[11].KeyID[15] := '3';
   Key[11].KeyID[16] := '2';
   Key[12].KeyID[1] := '0';
   Key[12].KeyID[2] := '3';
   Key[12].KeyID[3] := '7';
   Key[12].KeyID[4] := '2';
   Key[12].KeyID[5] := 'F';
   Key[12].KeyID[6] := '4';
   Key[12].KeyID[7] := 'D';
   Key[12].KeyID[8] := 'F';
   Key[12].KeyID[9] := '5';
   Key[12].KeyID[10] := 'C';
   Key[12].KeyID[11..12] := '0';
   Key[12].KeyID[13] := '1';
   Key[12].KeyID[14] := '0';
   Key[12].KeyID[15] := '3';
   Key[12].KeyID[16] := '2';
   Key[13].KeyID[1] := '0';
   Key[13].KeyID[2] := '3';
   Key[13].KeyID[3] := '7';
   Key[13].KeyID[4] := '2';
   Key[13].KeyID[5] := 'C';
   Key[13].KeyID[6] := '9';
   Key[13].KeyID[7] := '1';
   Key[13].KeyID[8..9] := '6';
   Key[13].KeyID[10] := '7';
   Key[13].KeyID[11..12] := '0';
   Key[13].KeyID[13] := '1';
   Key[13].KeyID[14] := '0';
   Key[13].KeyID[15] := '3';
   Key[13].KeyID[16] := '2';
   Key[14].KeyID[1] := '0';
   Key[14].KeyID[2] := '3';
   Key[14].KeyID[3] := '2';
   Key[14].KeyID[4] := '3';
   Key[14].KeyID[5] := 'C';
   Key[14].KeyID[6] := 'F';
   Key[14].KeyID[7] := '5';
   Key[14].KeyID[8] := 'E';
   Key[14].KeyID[9..10] := 'B';
   Key[14].KeyID[11..12] := '0';
   Key[14].KeyID[13] := '1';
   Key[14].KeyID[14] := '0';
   Key[14].KeyID[15] := '3';
   Key[14].KeyID[16] := '2';
   Key[15].KeyID[1] := '0';
   Key[15].KeyID[2] := '3';
   Key[15].KeyID[3] := '6';
   Key[15].KeyID[4] := '1';
   Key[15].KeyID[5] := 'E';
   Key[15].KeyID[6] := '8';
   Key[15].KeyID[7] := '1';
   Key[15].KeyID[8] := '4';
   Key[15].KeyID[9] := 'A';
   Key[15].KeyID[10] := 'E';
   Key[15].KeyID[11..12] := '0';
   Key[15].KeyID[13] := '1';
   Key[15].KeyID[14] := '0';
   Key[15].KeyID[15] := '3';
   Key[15].KeyID[16] := '2';
   Key[16].KeyID[1] := '0';
   Key[16].KeyID[2] := '3';
   Key[16].KeyID[3] := '7';
   Key[16].KeyID[4] := '1';
   Key[16].KeyID[5] := 'E';
   Key[16].KeyID[6] := 'D';
   Key[16].KeyID[7] := '1';
   Key[16].KeyID[8] := '2';
   Key[16].KeyID[9] := 'B';
   Key[16].KeyID[10] := '7';
   Key[16].KeyID[11..12] := '0';
   Key[16].KeyID[13] := '1';
   Key[16].KeyID[14] := '0';
   Key[16].KeyID[15] := '3';
   Key[16].KeyID[16] := '2';
   Key[17].KeyID[1] := '0';
   Key[17].KeyID[2] := '3';
   Key[17].KeyID[3] := '7';
   Key[17].KeyID[4] := '2';
   Key[17].KeyID[5] := 'F';
   Key[17].KeyID[6] := '5';
   Key[17].KeyID[7] := '2';
   Key[17].KeyID[8] := 'C';
   Key[17].KeyID[9] := '6';
   Key[17].KeyID[10] := '8';
   Key[17].KeyID[11..12] := '0';
   Key[17].KeyID[13] := '1';
   Key[17].KeyID[14] := '0';
   Key[17].KeyID[15] := '3';
   Key[17].KeyID[16] := '2';
   Key[18].KeyID[1] := '0';
   Key[18].KeyID[2] := '3';
   Key[18].KeyID[3] := '7';
   Key[18].KeyID[4] := '1';
   Key[18].KeyID[5..7] := 'F';
   Key[18].KeyID[8] := 'C';
   Key[18].KeyID[9] := '4';
   Key[18].KeyID[10] := '2';
   Key[18].KeyID[11..12] := '0';
   Key[18].KeyID[13] := '1';
   Key[18].KeyID[14] := '0';
   Key[18].KeyID[15] := '3';
   Key[18].KeyID[16] := '2';
   Key[19].KeyID[1..16] := ' ';
   Key[20].KeyID[1..16] := ' ';
   Key[21].KeyID[1..16] := ' ';
   Key[22].KeyID[1..16] := ' ';
   Key[23].KeyID[1..16] := ' ';
   Key[24].KeyID[1..16] := ' ';
   Key[25].KeyID[1..16] := ' ';
   Key[26].KeyID[1..16] := ' ';
   Key[27].KeyID[1..16] := ' ';
   Key[28].KeyID[1..16] := ' ';
   Key[29].KeyID[1..16] := ' ';
   Key[30].KeyID[1..16] := ' ';
   Key[31].KeyID[1..16] := ' ';
   Key[32].KeyID[1..16] := ' ';
   Key[33].KeyID[1..16] := ' ';
   Key[34].KeyID[1..16] := ' ';
   Key[35].KeyID[1..16] := ' ';
   Key[36].KeyID[1..16] := ' ';
   Key[37].KeyID[1..16] := ' ';
   Key[38].KeyID[1..16] := ' ';
   Key[39].KeyID[1..16] := ' ';
   Key[40].KeyID[1..16] := ' ';
   Key[41].KeyID[1..16] := ' ';
   Key[42].KeyID[1..16] := ' ';
   Key[43].KeyID[1..16] := ' ';
   Key[44].KeyID[1..16] := ' ';
   Key[45].KeyID[1..16] := ' ';
   Key[46].KeyID[1..16] := ' ';
   Key[47].KeyID[1..16] := ' ';
   Key[48].KeyID[1..16] := ' ';
   Key[49].KeyID[1..16] := ' ';
   Key[50].KeyID[1..16] := ' ';
   Key[51].KeyID[1..16] := ' ';
   Key[52].KeyID[1..16] := ' ';
   Key[53].KeyID[1..16] := ' ';
   Key[54].KeyID[1..16] := ' ';
   Key[55].KeyID[1..16] := ' ';
   Key[56].KeyID[1..16] := ' ';
   Key[57].KeyID[1..16] := ' ';
   Key[58].KeyID[1..16] := ' ';
   Key[59].KeyID[1..16] := ' ';
   Key[60].KeyID[1..16] := ' ';
   Key[61].KeyID[1..16] := ' ';
   Key[62].KeyID[1..16] := ' ';
   Key[63].KeyID[1..16] := ' ';
   Key[64].KeyID[1..16] := ' ';
   Key[65].KeyID[1..16] := ' ';
   Key[66].KeyID[1..16] := ' ';
   Key[67].KeyID[1..16] := ' ';
   Key[68].KeyID[1..16] := ' ';
   Key[69].KeyID[1..16] := ' ';
   Key[70].KeyID[1..16] := ' ';
   Key[71].KeyID[1..16] := ' ';
   Key[72].KeyID[1..16] := ' ';
   Key[73].KeyID[1..16] := ' ';
   Key[74].KeyID[1..16] := ' ';
   Key[75].KeyID[1..16] := ' ';
   Key[76].KeyID[1..16] := ' ';
   Key[77].KeyID[1..16] := ' ';
   Key[78].KeyID[1..16] := ' ';
   Key[79].KeyID[1..16] := ' ';
   Key[80].KeyID[1..16] := ' ';
   Key[81].KeyID[1..16] := ' ';
   Key[82].KeyID[1..16] := ' ';
   Key[83].KeyID[1..16] := ' ';
   Key[84].KeyID[1..16] := ' ';
   Key[85].KeyID[1..16] := ' ';
   Key[86].KeyID[1..16] := ' ';
   Key[87].KeyID[1..16] := ' ';
   Key[88].KeyID[1..16] := ' ';
   Key[89].KeyID[1..16] := ' ';
   Key[90].KeyID[1..16] := ' ';
   Key[91].KeyID[1..16] := ' ';
   Key[92].KeyID[1..16] := ' ';
   Key[93].KeyID[1..16] := ' ';
   Key[94].KeyID[1..16] := ' ';
   Key[95].KeyID[1..16] := ' ';
   Key[96].KeyID[1..16] := ' ';
   Key[97].KeyID[1..16] := ' ';
   Key[98].KeyID[1..16] := ' ';
   Key[99].KeyID[1..16] := ' ';
   Key[100].KeyID[1..16] := ' ';
   Key[1].Comment[1..20] := ' ';
   Key[2].Comment[1..20] := ' ';
   Key[3].Comment[1..20] := ' ';
   Key[4].Comment[1..20] := ' ';
   Key[5].Comment[1..20] := ' ';
   Key[6].Comment[1..20] := ' ';
   Key[7].Comment[1..20] := ' ';
   Key[8].Comment[1..20] := ' ';
   Key[9].Comment[1..20] := ' ';
   Key[10].Comment[1..20] := ' ';
   Key[11].Comment[1..20] := ' ';
   Key[12].Comment[1..20] := ' ';
   Key[13].Comment[1..20] := ' ';
   Key[14].Comment[1..20] := ' ';
   Key[15].Comment[1..20] := ' ';
   Key[16].Comment[1..20] := ' ';
   Key[17].Comment[1..20] := ' ';
   Key[18].Comment[1..20] := ' ';
   Key[19].Comment[1..20] := ' ';
   Key[20].Comment[1..20] := ' ';
   Key[21].Comment[1..20] := ' ';
   Key[22].Comment[1..20] := ' ';
   Key[23].Comment[1..20] := ' ';
   Key[24].Comment[1..20] := ' ';
   Key[25].Comment[1..20] := ' ';
   Key[26].Comment[1..20] := ' ';
   Key[27].Comment[1..20] := ' ';
   Key[28].Comment[1..20] := ' ';
   Key[29].Comment[1..20] := ' ';
   Key[30].Comment[1..20] := ' ';
   Key[31].Comment[1..20] := ' ';
   Key[32].Comment[1..20] := ' ';
   Key[33].Comment[1..20] := ' ';
   Key[34].Comment[1..20] := ' ';
   Key[35].Comment[1..20] := ' ';
   Key[36].Comment[1..20] := ' ';
   Key[37].Comment[1..20] := ' ';
   Key[38].Comment[1..20] := ' ';
   Key[39].Comment[1..20] := ' ';
   Key[40].Comment[1..20] := ' ';
   Key[41].Comment[1..20] := ' ';
   Key[42].Comment[1..20] := ' ';
   Key[43].Comment[1..20] := ' ';
   Key[44].Comment[1..20] := ' ';
   Key[45].Comment[1..20] := ' ';
   Key[46].Comment[1..20] := ' ';
   Key[47].Comment[1..20] := ' ';
   Key[48].Comment[1..20] := ' ';
   Key[49].Comment[1..20] := ' ';
   Key[50].Comment[1..20] := ' ';
   Key[51].Comment[1..20] := ' ';
   Key[52].Comment[1..20] := ' ';
   Key[53].Comment[1..20] := ' ';
   Key[54].Comment[1..20] := ' ';
   Key[55].Comment[1..20] := ' ';
   Key[56].Comment[1..20] := ' ';
   Key[57].Comment[1..20] := ' ';
   Key[58].Comment[1..20] := ' ';
   Key[59].Comment[1..20] := ' ';
   Key[60].Comment[1..20] := ' ';
   Key[61].Comment[1..20] := ' ';
   Key[62].Comment[1..20] := ' ';
   Key[63].Comment[1..20] := ' ';
   Key[64].Comment[1..20] := ' ';
   Key[65].Comment[1..20] := ' ';
   Key[66].Comment[1..20] := ' ';
   Key[67].Comment[1..20] := ' ';
   Key[68].Comment[1..20] := ' ';
   Key[69].Comment[1..20] := ' ';
   Key[70].Comment[1..20] := ' ';
   Key[71].Comment[1..20] := ' ';
   Key[72].Comment[1..20] := ' ';
   Key[73].Comment[1..20] := ' ';
   Key[74].Comment[1..20] := ' ';
   Key[75].Comment[1..20] := ' ';
   Key[76].Comment[1..20] := ' ';
   Key[77].Comment[1..20] := ' ';
   Key[78].Comment[1..20] := ' ';
   Key[79].Comment[1..20] := ' ';
   Key[80].Comment[1..20] := ' ';
   Key[81].Comment[1..20] := ' ';
   Key[82].Comment[1..20] := ' ';
   Key[83].Comment[1..20] := ' ';
   Key[84].Comment[1..20] := ' ';
   Key[85].Comment[1..20] := ' ';
   Key[86].Comment[1..20] := ' ';
   Key[87].Comment[1..20] := ' ';
   Key[88].Comment[1..20] := ' ';
   Key[89].Comment[1..20] := ' ';
   Key[90].Comment[1..20] := ' ';
   Key[91].Comment[1..20] := ' ';
   Key[92].Comment[1..20] := ' ';
   Key[93].Comment[1..20] := ' ';
   Key[94].Comment[1..20] := ' ';
   Key[95].Comment[1..20] := ' ';
   Key[96].Comment[1..20] := ' ';
   Key[97].Comment[1..20] := ' ';
   Key[98].Comment[1..20] := ' ';
   Key[99].Comment[1..20] := ' ';
   Key[100].Comment[1..20] := ' ';
END_DATA_BLOCK

DATA_BLOCK "HMIData"   // DB1
{ S7_Optimized_Access := 'TRUE' }
VERSION : 0.1
// stored: AutoNumber false, DBAccessibleFromOPCUA true, DBAccessibleFromWebserver true, IsOnlyStoredInLoadMemory false, IsRetainMemResEnabled false, IsWriteProtectedInAS false, MemoryReserve 100
   VAR
      HMI { S7_SetPoint := 'True'} : "UDT_HMI";
      ManualCommandHMI : Int := 0;
      ManualCommand : Int := 0;
   END_VAR
BEGIN
   HMI.ScreenData[1..5] := 16#0000;
   HMI.UserNumber := 0;
   HMI.ActualScreenNumber := 0;
   HMI.RequiredScreenNumber := 0;
   HMI.FunctionKeys[1..8] := FALSE;
END_DATA_BLOCK

DATA_BLOCK "SystemHMI"   // DB10
{ S7_Optimized_Access := 'TRUE' }
VERSION : 0.1
// stored: AutoNumber false, DBAccessibleFromOPCUA true, DBAccessibleFromWebserver true, IsOnlyStoredInLoadMemory false, IsRetainMemResEnabled false, IsWriteProtectedInAS false, MemoryReserve 100
   VAR
      AlarmActive : Bool := FALSE;
      AlarmActiveBlinking : Bool := FALSE;
      WarningActive : Bool := FALSE;
      BasicPosition : Bool := FALSE;
      GoToBasicPosition : Bool := FALSE;
      ManualMode : Bool := TRUE;
      AutomaticMode : Bool := FALSE;
      ManualCommand : Int := 0;
      BasicPositionMessage : Int := 0;
      BasicPositionStep : Int := 0;
      ManualFromRobot : Bool := FALSE;
      HydraulicPumpAutoControl : Bool := FALSE;
      BasicPositionSt1 : Bool := FALSE;
      BasicPositionSt2 : Bool := FALSE;
      BasicPositionFitting : Bool := FALSE;
      BasicPositionGripper1 : Bool := FALSE;
      BasicPositionStartHMI : Bool := FALSE;
      AutoStartHMI : Bool := FALSE;
      ResetPartsErrors : Bool := FALSE;
      ModeChanged : Bool := FALSE;
   END_VAR
BEGIN
END_DATA_BLOCK

DATA_BLOCK "db_REC_IJCORE"   // DB1006
{ S7_Optimized_Access := 'FALSE' }
VERSION : 0.1
// stored: AutoNumber false, DBAccessibleFromOPCUA true, DBAccessibleFromWebserver true, IsOnlyStoredInLoadMemory false, IsWriteProtectedInAS false
   VAR
      SW_Message : Array[1..300] of Word;
      Message : Array[1..100] of Struct
         Answer : Int;
         Content : Array[1..30] of Byte;
      END_STRUCT;
   END_VAR
BEGIN
END_DATA_BLOCK

DATA_BLOCK "db_SEND_IJCORE"   // DB1005
{ S7_Optimized_Access := 'FALSE' }
VERSION : 0.1
// stored: AutoNumber false, DBAccessibleFromOPCUA true, DBAccessibleFromWebserver true, IsOnlyStoredInLoadMemory false, IsWriteProtectedInAS false
   VAR
      Awake_DW : Word;
      Awake_SW : Int;
      SW_Message : Array[1..300] of Word;
      Message : Array[1..100] of Struct
         Content : Array[1..80] of Byte;
      END_STRUCT;
   END_VAR
BEGIN
END_DATA_BLOCK

DATA_BLOCK "StationParameters"   // DB9
{ S7_Optimized_Access := 'TRUE' }
VERSION : 0.1
// stored: AutoNumber true, DBAccessibleFromOPCUA true, DBAccessibleFromWebserver true, IsOnlyStoredInLoadMemory false, IsRetainMemResEnabled false, IsWriteProtectedInAS false, MemoryReserve 100
   VAR RETAIN
      PumpStopDelay : Time := T#2S;
      ReleasePressureDelay : Time := T#5S;
      VH1BasicPositionMin : Real := -5.0;
      VH1BasicPositionMax : Real := 10.0;
      VH2BasicPositionMin : Real := -5.0;
      VH2BasicPositionMax : Real := 10.0;
      DisableScanner : Bool := TRUE;
      NOKBoxSize : Int := 3;
      OKUpperStockSize : Int := 3;
      OKLowerStockSize : Int := 3;
      GhostMode : Bool := FALSE;
      VH1MaxPosition : Real := 63.0;
      VH2MaxPosition : Real := 63.0;
      MaximalFittingTime : Time := T#20S;
      DisableR1Detection1 : Bool := FALSE;
      DisableR1Detection2 : Bool := FALSE;
      ManipulatorTimeBeforeLowerFixation : Time := T#5S;
      HangerDetectionORfunction : Bool := FALSE;
      AudioSignalizationTimeBeforeSafety : Time := T#5S;
      Servo : "UDT_ServoPrameters";
      ServoPositions { S7_SetPoint := 'True'} : Array[0..9] of DInt;
      DontUseHangerForParts { S7_SetPoint := 'True'} : Bool := TRUE;
      ManipulatorCommOff { S7_SetPoint := 'True'} : Bool := TRUE;
   END_VAR
BEGIN
   Servo.Velocity := 500;
   Servo.OverV := 100;
   Servo.OverAcc := 50;
   Servo.OverDec := 100;
   ServoPositions[0] := 10002;
   ServoPositions[1] := 784500;
   ServoPositions[2] := 1510500;
   ServoPositions[3..9] := 0;
END_DATA_BLOCK

DATA_BLOCK "DB_ProductionCountersEdit"   // DB66
{ S7_Optimized_Access := 'TRUE' }
VERSION : 0.1
// stored: AutoNumber true, DBAccessibleFromOPCUA true, DBAccessibleFromWebserver true, IsOnlyStoredInLoadMemory false, IsRetainMemResEnabled false, IsWriteProtectedInAS false, MemoryReserve 100
   VAR
      ProgramNumber : Int := 1;
      ProgramName : String[50] := '2569703X-LH';
      ProductCounters { S7_SetPoint := 'True'} : "UDT_ProductionProgramCounters";
      SettingsCanBeChanged : Bool := FALSE;
      DeleteCounters : Int := 0;
   END_VAR
BEGIN
   ProductCounters.Product[1].Shift[1..3].Ok := 0;
   ProductCounters.Product[2].Shift[1..3].Ok := 0;
   ProductCounters.Product[3].Shift[1..3].Ok := 0;
   ProductCounters.Product[4].Shift[1..3].Ok := 0;
   ProductCounters.Product[5].Shift[1..3].Ok := 0;
   ProductCounters.Product[6].Shift[1..3].Ok := 0;
   ProductCounters.Product[7].Shift[1..3].Ok := 0;
   ProductCounters.Product[8].Shift[1..3].Ok := 0;
   ProductCounters.Product[1].Shift[1..3].Nok := 0;
   ProductCounters.Product[2].Shift[1..3].Nok := 0;
   ProductCounters.Product[3].Shift[1..3].Nok := 0;
   ProductCounters.Product[4].Shift[1..3].Nok := 0;
   ProductCounters.Product[5].Shift[1..3].Nok := 0;
   ProductCounters.Product[6].Shift[1..3].Nok := 0;
   ProductCounters.Product[7].Shift[1..3].Nok := 0;
   ProductCounters.Product[8].Shift[1..3].Nok := 0;
   ProductCounters.Product[1..8].Overall.Ok := 0;
   ProductCounters.Product[1..8].Overall.Nok := 0;
END_DATA_BLOCK

DATA_BLOCK "DB_ProductionCountersList"   // DB65
{ S7_Optimized_Access := 'TRUE' }
VERSION : 0.1
// stored: AutoNumber true, DBAccessibleFromOPCUA true, DBAccessibleFromWebserver true, IsOnlyStoredInLoadMemory false, IsRetainMemResEnabled false, IsWriteProtectedInAS false, MemoryReserve 100
   VAR RETAIN
      Program { S7_SetPoint := 'True'} : Array[1.."NumberOfProductionPrograms"] of "UDT_ProductionProgramCounters";
      Machine : "UDT_Counters";
   END_VAR
BEGIN
   Program[1].Product[1].Shift[1..3].Ok := 0;
   Program[1].Product[2].Shift[1..3].Ok := 0;
   Program[1].Product[3].Shift[1..3].Ok := 0;
   Program[1].Product[4].Shift[1..3].Ok := 0;
   Program[1].Product[5].Shift[1..3].Ok := 0;
   Program[1].Product[6].Shift[1..3].Ok := 0;
   Program[1].Product[7].Shift[1..3].Ok := 0;
   Program[1].Product[8].Shift[1..3].Ok := 0;
   Program[2].Product[1].Shift[1..3].Ok := 0;
   Program[2].Product[2].Shift[1..3].Ok := 0;
   Program[2].Product[3].Shift[1..3].Ok := 0;
   Program[2].Product[4].Shift[1..3].Ok := 0;
   Program[2].Product[5].Shift[1..3].Ok := 0;
   Program[2].Product[6].Shift[1..3].Ok := 0;
   Program[2].Product[7].Shift[1..3].Ok := 0;
   Program[2].Product[8].Shift[1..3].Ok := 0;
   Program[3].Product[1].Shift[1..3].Ok := 0;
   Program[3].Product[2].Shift[1..3].Ok := 0;
   Program[3].Product[3].Shift[1..3].Ok := 0;
   Program[3].Product[4].Shift[1..3].Ok := 0;
   Program[3].Product[5].Shift[1..3].Ok := 0;
   Program[3].Product[6].Shift[1..3].Ok := 0;
   Program[3].Product[7].Shift[1..3].Ok := 0;
   Program[3].Product[8].Shift[1..3].Ok := 0;
   Program[4].Product[1].Shift[1..3].Ok := 0;
   Program[4].Product[2].Shift[1..3].Ok := 0;
   Program[4].Product[3].Shift[1..3].Ok := 0;
   Program[4].Product[4].Shift[1..3].Ok := 0;
   Program[4].Product[5].Shift[1..3].Ok := 0;
   Program[4].Product[6].Shift[1..3].Ok := 0;
   Program[4].Product[7].Shift[1..3].Ok := 0;
   Program[4].Product[8].Shift[1..3].Ok := 0;
   Program[5].Product[1].Shift[1..3].Ok := 0;
   Program[5].Product[2].Shift[1..3].Ok := 0;
   Program[5].Product[3].Shift[1..3].Ok := 0;
   Program[5].Product[4].Shift[1..3].Ok := 0;
   Program[5].Product[5].Shift[1..3].Ok := 0;
   Program[5].Product[6].Shift[1..3].Ok := 0;
   Program[5].Product[7].Shift[1..3].Ok := 0;
   Program[5].Product[8].Shift[1..3].Ok := 0;
   Program[6].Product[1].Shift[1..3].Ok := 0;
   Program[6].Product[2].Shift[1..3].Ok := 0;
   Program[6].Product[3].Shift[1..3].Ok := 0;
   Program[6].Product[4].Shift[1..3].Ok := 0;
   Program[6].Product[5].Shift[1..3].Ok := 0;
   Program[6].Product[6].Shift[1..3].Ok := 0;
   Program[6].Product[7].Shift[1..3].Ok := 0;
   Program[6].Product[8].Shift[1..3].Ok := 0;
   Program[7].Product[1].Shift[1..3].Ok := 0;
   Program[7].Product[2].Shift[1..3].Ok := 0;
   Program[7].Product[3].Shift[1..3].Ok := 0;
   Program[7].Product[4].Shift[1..3].Ok := 0;
   Program[7].Product[5].Shift[1..3].Ok := 0;
   Program[7].Product[6].Shift[1..3].Ok := 0;
   Program[7].Product[7].Shift[1..3].Ok := 0;
   Program[7].Product[8].Shift[1..3].Ok := 0;
   Program[8].Product[1].Shift[1..3].Ok := 0;
   Program[8].Product[2].Shift[1..3].Ok := 0;
   Program[8].Product[3].Shift[1..3].Ok := 0;
   Program[8].Product[4].Shift[1..3].Ok := 0;
   Program[8].Product[5].Shift[1..3].Ok := 0;
   Program[8].Product[6].Shift[1..3].Ok := 0;
   Program[8].Product[7].Shift[1..3].Ok := 0;
   Program[8].Product[8].Shift[1..3].Ok := 0;
   Program[1].Product[1].Shift[1..3].Nok := 0;
   Program[1].Product[2].Shift[1..3].Nok := 0;
   Program[1].Product[3].Shift[1..3].Nok := 0;
   Program[1].Product[4].Shift[1..3].Nok := 0;
   Program[1].Product[5].Shift[1..3].Nok := 0;
   Program[1].Product[6].Shift[1..3].Nok := 0;
   Program[1].Product[7].Shift[1..3].Nok := 0;
   Program[1].Product[8].Shift[1..3].Nok := 0;
   Program[2].Product[1].Shift[1..3].Nok := 0;
   Program[2].Product[2].Shift[1..3].Nok := 0;
   Program[2].Product[3].Shift[1..3].Nok := 0;
   Program[2].Product[4].Shift[1..3].Nok := 0;
   Program[2].Product[5].Shift[1..3].Nok := 0;
   Program[2].Product[6].Shift[1..3].Nok := 0;
   Program[2].Product[7].Shift[1..3].Nok := 0;
   Program[2].Product[8].Shift[1..3].Nok := 0;
   Program[3].Product[1].Shift[1..3].Nok := 0;
   Program[3].Product[2].Shift[1..3].Nok := 0;
   Program[3].Product[3].Shift[1..3].Nok := 0;
   Program[3].Product[4].Shift[1..3].Nok := 0;
   Program[3].Product[5].Shift[1..3].Nok := 0;
   Program[3].Product[6].Shift[1..3].Nok := 0;
   Program[3].Product[7].Shift[1..3].Nok := 0;
   Program[3].Product[8].Shift[1..3].Nok := 0;
   Program[4].Product[1].Shift[1..3].Nok := 0;
   Program[4].Product[2].Shift[1..3].Nok := 0;
   Program[4].Product[3].Shift[1..3].Nok := 0;
   Program[4].Product[4].Shift[1..3].Nok := 0;
   Program[4].Product[5].Shift[1..3].Nok := 0;
   Program[4].Product[6].Shift[1..3].Nok := 0;
   Program[4].Product[7].Shift[1..3].Nok := 0;
   Program[4].Product[8].Shift[1..3].Nok := 0;
   Program[5].Product[1].Shift[1..3].Nok := 0;
   Program[5].Product[2].Shift[1..3].Nok := 0;
   Program[5].Product[3].Shift[1..3].Nok := 0;
   Program[5].Product[4].Shift[1..3].Nok := 0;
   Program[5].Product[5].Shift[1..3].Nok := 0;
   Program[5].Product[6].Shift[1..3].Nok := 0;
   Program[5].Product[7].Shift[1..3].Nok := 0;
   Program[5].Product[8].Shift[1..3].Nok := 0;
   Program[6].Product[1].Shift[1..3].Nok := 0;
   Program[6].Product[2].Shift[1..3].Nok := 0;
   Program[6].Product[3].Shift[1..3].Nok := 0;
   Program[6].Product[4].Shift[1..3].Nok := 0;
   Program[6].Product[5].Shift[1..3].Nok := 0;
   Program[6].Product[6].Shift[1..3].Nok := 0;
   Program[6].Product[7].Shift[1..3].Nok := 0;
   Program[6].Product[8].Shift[1..3].Nok := 0;
   Program[7].Product[1].Shift[1..3].Nok := 0;
   Program[7].Product[2].Shift[1..3].Nok := 0;
   Program[7].Product[3].Shift[1..3].Nok := 0;
   Program[7].Product[4].Shift[1..3].Nok := 0;
   Program[7].Product[5].Shift[1..3].Nok := 0;
   Program[7].Product[6].Shift[1..3].Nok := 0;
   Program[7].Product[7].Shift[1..3].Nok := 0;
   Program[7].Product[8].Shift[1..3].Nok := 0;
   Program[8].Product[1].Shift[1..3].Nok := 0;
   Program[8].Product[2].Shift[1..3].Nok := 0;
   Program[8].Product[3].Shift[1..3].Nok := 0;
   Program[8].Product[4].Shift[1..3].Nok := 0;
   Program[8].Product[5].Shift[1..3].Nok := 0;
   Program[8].Product[6].Shift[1..3].Nok := 0;
   Program[8].Product[7].Shift[1..3].Nok := 0;
   Program[8].Product[8].Shift[1..3].Nok := 0;
   Program[1].Product[1].Overall.Ok := 62;
   Program[1].Product[2..8].Overall.Ok := 0;
   Program[2].Product[1].Overall.Ok := 32;
   Program[2].Product[2..8].Overall.Ok := 0;
   Program[3].Product[1..8].Overall.Ok := 0;
   Program[4].Product[1..8].Overall.Ok := 0;
   Program[5].Product[1].Overall.Ok := 141;
   Program[5].Product[2..8].Overall.Ok := 0;
   Program[6].Product[1].Overall.Ok := 40;
   Program[6].Product[2..8].Overall.Ok := 0;
   Program[7].Product[1].Overall.Ok := 50;
   Program[7].Product[2..8].Overall.Ok := 0;
   Program[8].Product[1..8].Overall.Ok := 0;
   Program[1].Product[1].Overall.Nok := 9;
   Program[1].Product[2..8].Overall.Nok := 0;
   Program[2].Product[1].Overall.Nok := 7;
   Program[2].Product[2..8].Overall.Nok := 0;
   Program[3].Product[1..8].Overall.Nok := 0;
   Program[4].Product[1..8].Overall.Nok := 0;
   Program[5].Product[1].Overall.Nok := 43;
   Program[5].Product[2..8].Overall.Nok := 0;
   Program[6].Product[1].Overall.Nok := 3;
   Program[6].Product[2..8].Overall.Nok := 0;
   Program[7].Product[1..8].Overall.Nok := 0;
   Program[8].Product[1..8].Overall.Nok := 0;
   Machine.Ok := 325;
   Machine.Nok := 62;
END_DATA_BLOCK

DATA_BLOCK "DB_ProductionProgramActual"   // DB6101
{ S7_Optimized_Access := 'TRUE' }
VERSION : 0.1
// stored: AutoNumber false, DBAccessibleFromOPCUA true, DBAccessibleFromWebserver true, IsOnlyStoredInLoadMemory false, IsRetainMemResEnabled false, IsWriteProtectedInAS false, MemoryReserve 100
   VAR
      Program { S7_SetPoint := 'True'} : "UDT_ProductionProgram";
      ProgrammNumber { S7_SetPoint := 'True'} : Int := 5;
      Load : Bool := FALSE;
      Save : Bool := FALSE;
      CanBeChanged : Bool := FALSE;
   END_VAR
BEGIN
   Program."Name" := 'startup';
   Program.CupformingParametersLeft.DigiforceProgram := 1;
   Program.CupformingParametersLeft.FinalSpeed := 25.0;
   Program.CupformingParametersLeft.ApproachSpeed := 25.0;
   Program.CupformingParametersLeft.FinalForce := 10.0;
   Program.CupformingParametersLeft.ApproachForce := 10.0;
   Program.CupformingParametersLeft.EndWayImmediate := 2.55;
   Program.CupformingParametersLeft.EndWayWithTimeout := 3.0;
   Program.CupformingParametersLeft.SwitchingWay := 20.0;
   Program.CupformingParametersLeft.EndWayTimeout := T#300MS;
   Program.CupformingParametersRight.DigiforceProgram := 1;
   Program.CupformingParametersRight.FinalSpeed := 25.0;
   Program.CupformingParametersRight.ApproachSpeed := 25.0;
   Program.CupformingParametersRight.FinalForce := 10.0;
   Program.CupformingParametersRight.ApproachForce := 10.0;
   Program.CupformingParametersRight.EndWayImmediate := 2.7;
   Program.CupformingParametersRight.EndWayWithTimeout := 3.0;
   Program.CupformingParametersRight.SwitchingWay := 20.0;
   Program.CupformingParametersRight.EndWayTimeout := T#300MS;
   Program.St1Insertion[1] := TRUE;
   Program.St1Insertion[2] := FALSE;
   Program.St1Insertion[3..5] := TRUE;
   Program.St1Insertion[6] := FALSE;
   Program.St1Insertion[7] := TRUE;
   Program.St1Insertion[8] := FALSE;
   Program.St1Insertion[9..10] := TRUE;
   Program.St1Insertion[11] := FALSE;
   Program.St1Insertion[12..17] := TRUE;
   Program.St1Insertion[18] := FALSE;
   Program.St1Insertion[19] := TRUE;
   Program.St1Insertion[20] := FALSE;
   Program.St1InsertionUsed[1..7] := TRUE;
   Program.St1InsertionUsed[8] := FALSE;
   Program.St1InsertionUsed[9..19] := TRUE;
   Program.St1InsertionUsed[20] := FALSE;
   Program.FaureciaNumber := '2567208X';
   Program.FaureciaNumberStartChar := 9;
   Program.FaureciaNumberLength := 8;
   Program.MechanicalType := 0;
END_DATA_BLOCK

DATA_BLOCK "DB_ProductionProgramEdit"   // DB6103
{ S7_Optimized_Access := 'FALSE' }
VERSION : 0.1
// stored: AutoNumber false, DBAccessibleFromOPCUA true, DBAccessibleFromWebserver true, IsOnlyStoredInLoadMemory false, IsWriteProtectedInAS false
   VAR
      ProgramEmpty { S7_SetPoint := 'True'} : "UDT_ProductionProgram";
      ProgramInBox { S7_SetPoint := 'True'} : "UDT_ProductionProgram";
      ProgramEdit { S7_SetPoint := 'True'} : "UDT_ProductionProgram";
      Commands : Struct
         ProgramEdit : Struct
            Number : UInt := 5;
            NumberLast : UInt := 5;
            NumberChanged : Bool := FALSE;
            NumberInBox : UInt := 5;
            Commands : UInt := 0;   // 1= Load, 2= Save, 3= Copy, 4= Paste, 5= Delete
            LoadAll : Bool := FALSE;
            ProgramChanged : Bool := FALSE;
            SettingsCanBeChanged : Bool := TRUE;
            ChangeButtonsBlinking : Bool := FALSE;
            ChangeButtonsVisibility : Bool := FALSE;
            CommandsVisibility : Bool := TRUE;
         END_STRUCT;
         ProductEdit : Struct
            Number : UInt := 1;
            NumberLast : UInt := 1;
            NumberChanged : Bool := FALSE;
            Load : Bool := FALSE;
         END_STRUCT;
         PositionEdit : Struct
            Number : UInt := 1;
            NumberLast : UInt := 1;
            NumberChanged : Bool := FALSE;
            Load : Bool := FALSE;
         END_STRUCT;
      END_STRUCT;
   END_VAR
BEGIN
   ProgramEmpty."Name" := '';
   ProgramEmpty.CupformingParametersLeft.DigiforceProgram := 0;
   ProgramEmpty.CupformingParametersLeft.FinalSpeed := 0.0;
   ProgramEmpty.CupformingParametersLeft.ApproachSpeed := 0.0;
   ProgramEmpty.CupformingParametersLeft.FinalForce := 0.0;
   ProgramEmpty.CupformingParametersLeft.ApproachForce := 0.0;
   ProgramEmpty.CupformingParametersLeft.EndWayImmediate := 0.0;
   ProgramEmpty.CupformingParametersLeft.EndWayWithTimeout := 0.0;
   ProgramEmpty.CupformingParametersLeft.SwitchingWay := 0.0;
   ProgramEmpty.CupformingParametersLeft.EndWayTimeout := T#0MS;
   ProgramEmpty.CupformingParametersRight.DigiforceProgram := 0;
   ProgramEmpty.CupformingParametersRight.FinalSpeed := 0.0;
   ProgramEmpty.CupformingParametersRight.ApproachSpeed := 0.0;
   ProgramEmpty.CupformingParametersRight.FinalForce := 0.0;
   ProgramEmpty.CupformingParametersRight.ApproachForce := 0.0;
   ProgramEmpty.CupformingParametersRight.EndWayImmediate := 0.0;
   ProgramEmpty.CupformingParametersRight.EndWayWithTimeout := 0.0;
   ProgramEmpty.CupformingParametersRight.SwitchingWay := 0.0;
   ProgramEmpty.CupformingParametersRight.EndWayTimeout := T#0MS;
   ProgramEmpty.St1Insertion[1..20] := FALSE;
   ProgramEmpty.St1InsertionUsed[1..20] := FALSE;
   ProgramEmpty.FaureciaNumber := '';
   ProgramEmpty.FaureciaNumberStartChar := 0;
   ProgramEmpty.FaureciaNumberLength := 0;
   ProgramEmpty.MechanicalType := 0;
   ProgramInBox."Name" := 'startup';
   ProgramInBox.CupformingParametersLeft.DigiforceProgram := 1;
   ProgramInBox.CupformingParametersLeft.FinalSpeed := 25.0;
   ProgramInBox.CupformingParametersLeft.ApproachSpeed := 25.0;
   ProgramInBox.CupformingParametersLeft.FinalForce := 10.0;
   ProgramInBox.CupformingParametersLeft.ApproachForce := 10.0;
   ProgramInBox.CupformingParametersLeft.EndWayImmediate := 2.55;
   ProgramInBox.CupformingParametersLeft.EndWayWithTimeout := 3.0;
   ProgramInBox.CupformingParametersLeft.SwitchingWay := 20.0;
   ProgramInBox.CupformingParametersLeft.EndWayTimeout := T#300MS;
   ProgramInBox.CupformingParametersRight.DigiforceProgram := 1;
   ProgramInBox.CupformingParametersRight.FinalSpeed := 25.0;
   ProgramInBox.CupformingParametersRight.ApproachSpeed := 25.0;
   ProgramInBox.CupformingParametersRight.FinalForce := 60.0;
   ProgramInBox.CupformingParametersRight.ApproachForce := 10.0;
   ProgramInBox.CupformingParametersRight.EndWayImmediate := 2.7;
   ProgramInBox.CupformingParametersRight.EndWayWithTimeout := 3.0;
   ProgramInBox.CupformingParametersRight.SwitchingWay := 20.0;
   ProgramInBox.CupformingParametersRight.EndWayTimeout := T#300MS;
   ProgramInBox.St1Insertion[1] := TRUE;
   ProgramInBox.St1Insertion[2] := FALSE;
   ProgramInBox.St1Insertion[3..5] := TRUE;
   ProgramInBox.St1Insertion[6] := FALSE;
   ProgramInBox.St1Insertion[7] := TRUE;
   ProgramInBox.St1Insertion[8] := FALSE;
   ProgramInBox.St1Insertion[9..10] := TRUE;
   ProgramInBox.St1Insertion[11] := FALSE;
   ProgramInBox.St1Insertion[12..17] := TRUE;
   ProgramInBox.St1Insertion[18] := FALSE;
   ProgramInBox.St1Insertion[19] := TRUE;
   ProgramInBox.St1Insertion[20] := FALSE;
   ProgramInBox.St1InsertionUsed[1..7] := TRUE;
   ProgramInBox.St1InsertionUsed[8] := FALSE;
   ProgramInBox.St1InsertionUsed[9..19] := TRUE;
   ProgramInBox.St1InsertionUsed[20] := FALSE;
   ProgramInBox.FaureciaNumber := '2567208X';
   ProgramInBox.FaureciaNumberStartChar := 9;
   ProgramInBox.FaureciaNumberLength := 8;
   ProgramInBox.MechanicalType := 0;
   ProgramEdit."Name" := 'startup';
   ProgramEdit.CupformingParametersLeft.DigiforceProgram := 1;
   ProgramEdit.CupformingParametersLeft.FinalSpeed := 25.0;
   ProgramEdit.CupformingParametersLeft.ApproachSpeed := 25.0;
   ProgramEdit.CupformingParametersLeft.FinalForce := 10.0;
   ProgramEdit.CupformingParametersLeft.ApproachForce := 10.0;
   ProgramEdit.CupformingParametersLeft.EndWayImmediate := 2.55;
   ProgramEdit.CupformingParametersLeft.EndWayWithTimeout := 3.0;
   ProgramEdit.CupformingParametersLeft.SwitchingWay := 20.0;
   ProgramEdit.CupformingParametersLeft.EndWayTimeout := T#300MS;
   ProgramEdit.CupformingParametersRight.DigiforceProgram := 1;
   ProgramEdit.CupformingParametersRight.FinalSpeed := 25.0;
   ProgramEdit.CupformingParametersRight.ApproachSpeed := 25.0;
   ProgramEdit.CupformingParametersRight.FinalForce := 60.0;
   ProgramEdit.CupformingParametersRight.ApproachForce := 10.0;
   ProgramEdit.CupformingParametersRight.EndWayImmediate := 2.7;
   ProgramEdit.CupformingParametersRight.EndWayWithTimeout := 3.0;
   ProgramEdit.CupformingParametersRight.SwitchingWay := 20.0;
   ProgramEdit.CupformingParametersRight.EndWayTimeout := T#300MS;
   ProgramEdit.St1Insertion[1] := TRUE;
   ProgramEdit.St1Insertion[2] := FALSE;
   ProgramEdit.St1Insertion[3..5] := TRUE;
   ProgramEdit.St1Insertion[6] := FALSE;
   ProgramEdit.St1Insertion[7] := TRUE;
   ProgramEdit.St1Insertion[8] := FALSE;
   ProgramEdit.St1Insertion[9..10] := TRUE;
   ProgramEdit.St1Insertion[11] := FALSE;
   ProgramEdit.St1Insertion[12..17] := TRUE;
   ProgramEdit.St1Insertion[18] := FALSE;
   ProgramEdit.St1Insertion[19] := TRUE;
   ProgramEdit.St1Insertion[20] := FALSE;
   ProgramEdit.St1InsertionUsed[1..7] := TRUE;
   ProgramEdit.St1InsertionUsed[8] := FALSE;
   ProgramEdit.St1InsertionUsed[9..19] := TRUE;
   ProgramEdit.St1InsertionUsed[20] := FALSE;
   ProgramEdit.FaureciaNumber := '2567208X';
   ProgramEdit.FaureciaNumberStartChar := 9;
   ProgramEdit.FaureciaNumberLength := 8;
   ProgramEdit.MechanicalType := 0;
END_DATA_BLOCK

DATA_BLOCK "DB_ProductionProgramList"   // DB6100
{ S7_Optimized_Access := 'FALSE' }
VERSION : 0.1
// stored: AutoNumber false, DBAccessibleFromOPCUA true, DBAccessibleFromWebserver true, IsOnlyStoredInLoadMemory false, IsWriteProtectedInAS false
   VAR RETAIN
      Program { S7_SetPoint := 'True'} : Array[1.."NumberOfProductionPrograms"] of "UDT_ProductionProgram";
   END_VAR
BEGIN
   Program[1]."Name" := 'LH-6 way';
   Program[2]."Name" := 'RH-6 way';
   Program[3]."Name" := 'LH-4 way';
   Program[4]."Name" := 'RH-4 way';
   Program[5]."Name" := 'startup';
   Program[6]."Name" := 'startup RH';
   Program[7..8]."Name" := '';
   Program[1].CupformingParametersLeft.DigiforceProgram := 1;
   Program[2].CupformingParametersLeft.DigiforceProgram := 2;
   Program[3].CupformingParametersLeft.DigiforceProgram := 1;
   Program[4].CupformingParametersLeft.DigiforceProgram := 2;
   Program[5..6].CupformingParametersLeft.DigiforceProgram := 1;
   Program[7..8].CupformingParametersLeft.DigiforceProgram := 0;
   Program[1..2].CupformingParametersLeft.FinalSpeed := 30.0;
   Program[3].CupformingParametersLeft.FinalSpeed := 20.0;
   Program[4].CupformingParametersLeft.FinalSpeed := 30.0;
   Program[5].CupformingParametersLeft.FinalSpeed := 25.0;
   Program[6].CupformingParametersLeft.FinalSpeed := 20.0;
   Program[7..8].CupformingParametersLeft.FinalSpeed := 0.0;
   Program[1..2].CupformingParametersLeft.ApproachSpeed := 95.0;
   Program[3].CupformingParametersLeft.ApproachSpeed := 100.0;
   Program[4].CupformingParametersLeft.ApproachSpeed := 95.0;
   Program[5].CupformingParametersLeft.ApproachSpeed := 25.0;
   Program[6].CupformingParametersLeft.ApproachSpeed := 100.0;
   Program[7..8].CupformingParametersLeft.ApproachSpeed := 0.0;
   Program[1..4].CupformingParametersLeft.FinalForce := 90.0;
   Program[5].CupformingParametersLeft.FinalForce := 10.0;
   Program[6].CupformingParametersLeft.FinalForce := 90.0;
   Program[7..8].CupformingParametersLeft.FinalForce := 0.0;
   Program[1..4].CupformingParametersLeft.ApproachForce := 20.0;
   Program[5].CupformingParametersLeft.ApproachForce := 10.0;
   Program[6].CupformingParametersLeft.ApproachForce := 20.0;
   Program[7..8].CupformingParametersLeft.ApproachForce := 0.0;
   Program[1..4].CupformingParametersLeft.EndWayImmediate := 7.5;
   Program[5].CupformingParametersLeft.EndWayImmediate := 2.55;
   Program[6].CupformingParametersLeft.EndWayImmediate := 9.9;
   Program[7..8].CupformingParametersLeft.EndWayImmediate := 0.0;
   Program[1..4].CupformingParametersLeft.EndWayWithTimeout := 8.6;
   Program[5].CupformingParametersLeft.EndWayWithTimeout := 3.0;
   Program[6].CupformingParametersLeft.EndWayWithTimeout := 9.9;
   Program[7..8].CupformingParametersLeft.EndWayWithTimeout := 0.0;
   Program[1..4].CupformingParametersLeft.SwitchingWay := 50.0;
   Program[5].CupformingParametersLeft.SwitchingWay := 20.0;
   Program[6].CupformingParametersLeft.SwitchingWay := 50.0;
   Program[7..8].CupformingParametersLeft.SwitchingWay := 0.0;
   Program[1..5].CupformingParametersLeft.EndWayTimeout := T#300MS;
   Program[6].CupformingParametersLeft.EndWayTimeout := T#200MS;
   Program[7..8].CupformingParametersLeft.EndWayTimeout := T#0MS;
   Program[1].CupformingParametersRight.DigiforceProgram := 1;
   Program[2].CupformingParametersRight.DigiforceProgram := 2;
   Program[3].CupformingParametersRight.DigiforceProgram := 1;
   Program[4].CupformingParametersRight.DigiforceProgram := 2;
   Program[5..6].CupformingParametersRight.DigiforceProgram := 1;
   Program[7..8].CupformingParametersRight.DigiforceProgram := 0;
   Program[1..4].CupformingParametersRight.FinalSpeed := 30.0;
   Program[5].CupformingParametersRight.FinalSpeed := 25.0;
   Program[6].CupformingParametersRight.FinalSpeed := 20.0;
   Program[7..8].CupformingParametersRight.FinalSpeed := 0.0;
   Program[1..2].CupformingParametersRight.ApproachSpeed := 100.0;
   Program[3].CupformingParametersRight.ApproachSpeed := 95.0;
   Program[4].CupformingParametersRight.ApproachSpeed := 100.0;
   Program[5].CupformingParametersRight.ApproachSpeed := 25.0;
   Program[6].CupformingParametersRight.ApproachSpeed := 100.0;
   Program[7..8].CupformingParametersRight.ApproachSpeed := 0.0;
   Program[1..6].CupformingParametersRight.FinalForce := 60.0;
   Program[7..8].CupformingParametersRight.FinalForce := 0.0;
   Program[1..6].CupformingParametersRight.ApproachForce := 10.0;
   Program[7..8].CupformingParametersRight.ApproachForce := 0.0;
   Program[1..4].CupformingParametersRight.EndWayImmediate := 7.8;
   Program[5].CupformingParametersRight.EndWayImmediate := 2.7;
   Program[6].CupformingParametersRight.EndWayImmediate := 9.9;
   Program[7..8].CupformingParametersRight.EndWayImmediate := 0.0;
   Program[1..2].CupformingParametersRight.EndWayWithTimeout := 8.4;
   Program[3].CupformingParametersRight.EndWayWithTimeout := 8.6;
   Program[4].CupformingParametersRight.EndWayWithTimeout := 8.4;
   Program[5].CupformingParametersRight.EndWayWithTimeout := 3.0;
   Program[6].CupformingParametersRight.EndWayWithTimeout := 9.9;
   Program[7..8].CupformingParametersRight.EndWayWithTimeout := 0.0;
   Program[1..4].CupformingParametersRight.SwitchingWay := 50.0;
   Program[5].CupformingParametersRight.SwitchingWay := 20.0;
   Program[6].CupformingParametersRight.SwitchingWay := 50.0;
   Program[7..8].CupformingParametersRight.SwitchingWay := 0.0;
   Program[1..4].CupformingParametersRight.EndWayTimeout := T#1S;
   Program[5].CupformingParametersRight.EndWayTimeout := T#300MS;
   Program[6].CupformingParametersRight.EndWayTimeout := T#200MS;
   Program[7..8].CupformingParametersRight.EndWayTimeout := T#0MS;
   Program[1].St1Insertion[1..6] := TRUE;
   Program[1].St1Insertion[7..20] := FALSE;
   Program[2].St1Insertion[1..6] := TRUE;
   Program[2].St1Insertion[7..20] := FALSE;
   Program[3].St1Insertion[1..2] := TRUE;
   Program[3].St1Insertion[3] := FALSE;
   Program[3].St1Insertion[4..6] := TRUE;
   Program[3].St1Insertion[7..20] := FALSE;
   Program[4].St1Insertion[1..5] := TRUE;
   Program[4].St1Insertion[6..20] := FALSE;
   Program[5].St1Insertion[1] := TRUE;
   Program[5].St1Insertion[2] := FALSE;
   Program[5].St1Insertion[3..5] := TRUE;
   Program[5].St1Insertion[6] := FALSE;
   Program[5].St1Insertion[7] := TRUE;
   Program[5].St1Insertion[8] := FALSE;
   Program[5].St1Insertion[9..10] := TRUE;
   Program[5].St1Insertion[11] := FALSE;
   Program[5].St1Insertion[12..17] := TRUE;
   Program[5].St1Insertion[18] := FALSE;
   Program[5].St1Insertion[19] := TRUE;
   Program[5].St1Insertion[20] := FALSE;
   Program[6].St1Insertion[1..4] := TRUE;
   Program[6].St1Insertion[5..20] := FALSE;
   Program[7].St1Insertion[1..20] := FALSE;
   Program[8].St1Insertion[1..20] := FALSE;
   Program[1].St1InsertionUsed[1..6] := TRUE;
   Program[1].St1InsertionUsed[7..20] := FALSE;
   Program[2].St1InsertionUsed[1..6] := TRUE;
   Program[2].St1InsertionUsed[7..20] := FALSE;
   Program[3].St1InsertionUsed[1..2] := TRUE;
   Program[3].St1InsertionUsed[3] := FALSE;
   Program[3].St1InsertionUsed[4..6] := TRUE;
   Program[3].St1InsertionUsed[7..20] := FALSE;
   Program[4].St1InsertionUsed[1..5] := TRUE;
   Program[4].St1InsertionUsed[6..20] := FALSE;
   Program[5].St1InsertionUsed[1..7] := TRUE;
   Program[5].St1InsertionUsed[8] := FALSE;
   Program[5].St1InsertionUsed[9..19] := TRUE;
   Program[5].St1InsertionUsed[20] := FALSE;
   Program[6].St1InsertionUsed[1..4] := TRUE;
   Program[6].St1InsertionUsed[5..20] := FALSE;
   Program[7].St1InsertionUsed[1..20] := FALSE;
   Program[8].St1InsertionUsed[1..20] := FALSE;
   Program[1].FaureciaNumber := '2824317X';
   Program[2].FaureciaNumber := '2841135X';
   Program[3].FaureciaNumber := '2824317X';
   Program[4].FaureciaNumber := '2841135X';
   Program[5].FaureciaNumber := '2567208X';
   Program[6].FaureciaNumber := 'xxxx';
   Program[7..8].FaureciaNumber := '';
   Program[1..6].FaureciaNumberStartChar := 9;
   Program[7..8].FaureciaNumberStartChar := 0;
   Program[1..6].FaureciaNumberLength := 8;
   Program[7..8].FaureciaNumberLength := 0;
   Program[1].MechanicalType := 0;
   Program[2].MechanicalType := 1;
   Program[3].MechanicalType := 0;
   Program[4].MechanicalType := 1;
   Program[5].MechanicalType := 0;
   Program[6].MechanicalType := 1;
   Program[7..8].MechanicalType := 0;
   Program[1].Camera_program[0] := 0;
   Program[1].Camera_program[1..4] := 1;
   Program[2].Camera_program[0..4] := 0;
   Program[3].Camera_program[0] := 0;
   Program[3].Camera_program[1] := 1;
   Program[3].Camera_program[2..3] := 3;
   Program[3].Camera_program[4] := 1;
   Program[4].Camera_program[0..4] := 0;
   Program[5].Camera_program[0..4] := 0;
   Program[6].Camera_program[0..4] := 0;
   Program[7].Camera_program[0..1] := 0;
   Program[7].Camera_program[2..3] := 4;
   Program[7].Camera_program[4] := 0;
   Program[8].Camera_program[0..4] := 0;
   Program[1].Riveting_program_left[0] := 0;
   Program[1].Riveting_program_left[1..2] := 1;
   Program[2].Riveting_program_left[0] := 0;
   Program[2].Riveting_program_left[1] := 3;
   Program[2].Riveting_program_left[2] := 1;
   Program[3].Riveting_program_left[0] := 0;
   Program[3].Riveting_program_left[1] := 3;
   Program[3].Riveting_program_left[2] := 1;
   Program[4].Riveting_program_left[0] := 0;
   Program[4].Riveting_program_left[1] := 3;
   Program[4].Riveting_program_left[2] := 1;
   Program[5].Riveting_program_left[0..2] := 0;
   Program[6].Riveting_program_left[0] := 0;
   Program[6].Riveting_program_left[1..2] := 2;
   Program[7].Riveting_program_left[0..2] := 0;
   Program[8].Riveting_program_left[0..2] := 0;
   Program[1].Riveting_program_right[0] := 0;
   Program[1].Riveting_program_right[1..2] := 1;
   Program[2].Riveting_program_right[0] := 0;
   Program[2].Riveting_program_right[1..2] := 1;
   Program[3].Riveting_program_right[0] := 0;
   Program[3].Riveting_program_right[1] := 3;
   Program[3].Riveting_program_right[2] := 1;
   Program[4].Riveting_program_right[0] := 0;
   Program[4].Riveting_program_right[1] := 3;
   Program[4].Riveting_program_right[2] := 1;
   Program[5].Riveting_program_right[0..2] := 0;
   Program[6].Riveting_program_right[0] := 0;
   Program[6].Riveting_program_right[1..2] := 2;
   Program[7].Riveting_program_right[0..2] := 0;
   Program[8].Riveting_program_right[0..2] := 0;
   Program[1..2].Total_number_of_rivets_4 := TRUE;
   Program[3..5].Total_number_of_rivets_4 := FALSE;
   Program[6].Total_number_of_rivets_4 := TRUE;
   Program[7..8].Total_number_of_rivets_4 := FALSE;
   Program[1..8].NumberOfReadings := 0;
   Program[1].Readings[1..4].Enable := FALSE;
   Program[2].Readings[1..4].Enable := FALSE;
   Program[3].Readings[1..4].Enable := FALSE;
   Program[4].Readings[1..4].Enable := FALSE;
   Program[5].Readings[1..4].Enable := FALSE;
   Program[6].Readings[1..4].Enable := FALSE;
   Program[7].Readings[1..4].Enable := FALSE;
   Program[8].Readings[1..4].Enable := FALSE;
   Program[1].Readings[1..4].ReaderNumber := 0;
   Program[2].Readings[1..4].ReaderNumber := 0;
   Program[3].Readings[1..4].ReaderNumber := 0;
   Program[4].Readings[1..4].ReaderNumber := 0;
   Program[5].Readings[1..4].ReaderNumber := 0;
   Program[6].Readings[1..4].ReaderNumber := 0;
   Program[7].Readings[1..4].ReaderNumber := 0;
   Program[8].Readings[1..4].ReaderNumber := 0;
   Program[1].Readings[1..4]."Name" := WSTRING#'';
   Program[2].Readings[1..4]."Name" := WSTRING#'';
   Program[3].Readings[1..4]."Name" := WSTRING#'';
   Program[4].Readings[1..4]."Name" := WSTRING#'';
   Program[5].Readings[1..4]."Name" := WSTRING#'';
   Program[6].Readings[1..4]."Name" := WSTRING#'';
   Program[7].Readings[1..4]."Name" := WSTRING#'';
   Program[8].Readings[1..4]."Name" := WSTRING#'';
   Program[1].Readings[1..4].LabelType := 0;
   Program[2].Readings[1..4].LabelType := 0;
   Program[3].Readings[1..4].LabelType := 0;
   Program[4].Readings[1..4].LabelType := 0;
   Program[5].Readings[1..4].LabelType := 0;
   Program[6].Readings[1..4].LabelType := 0;
   Program[7].Readings[1..4].LabelType := 0;
   Program[8].Readings[1..4].LabelType := 0;
   Program[1].Readings[1..4].ReferenceToFound := WSTRING#'';
   Program[2].Readings[1..4].ReferenceToFound := WSTRING#'';
   Program[3].Readings[1..4].ReferenceToFound := WSTRING#'';
   Program[4].Readings[1..4].ReferenceToFound := WSTRING#'';
   Program[5].Readings[1..4].ReferenceToFound := WSTRING#'';
   Program[6].Readings[1..4].ReferenceToFound := WSTRING#'';
   Program[7].Readings[1..4].ReferenceToFound := WSTRING#'';
   Program[8].Readings[1..4].ReferenceToFound := WSTRING#'';
   Program[1].Readings[1..4].ReferenceStartPosition := 0;
   Program[2].Readings[1..4].ReferenceStartPosition := 0;
   Program[3].Readings[1..4].ReferenceStartPosition := 0;
   Program[4].Readings[1..4].ReferenceStartPosition := 0;
   Program[5].Readings[1..4].ReferenceStartPosition := 0;
   Program[6].Readings[1..4].ReferenceStartPosition := 0;
   Program[7].Readings[1..4].ReferenceStartPosition := 0;
   Program[8].Readings[1..4].ReferenceStartPosition := 0;
   Program[1].Readings[1..4].ReferenceLenght := 0;
   Program[2].Readings[1..4].ReferenceLenght := 0;
   Program[3].Readings[1..4].ReferenceLenght := 0;
   Program[4].Readings[1..4].ReferenceLenght := 0;
   Program[5].Readings[1..4].ReferenceLenght := 0;
   Program[6].Readings[1..4].ReferenceLenght := 0;
   Program[7].Readings[1..4].ReferenceLenght := 0;
   Program[8].Readings[1..4].ReferenceLenght := 0;
   Program[1].Readings[1..4].MasterReadingNumber := 0;
   Program[2].Readings[1..4].MasterReadingNumber := 0;
   Program[3].Readings[1..4].MasterReadingNumber := 0;
   Program[4].Readings[1..4].MasterReadingNumber := 0;
   Program[5].Readings[1..4].MasterReadingNumber := 0;
   Program[6].Readings[1..4].MasterReadingNumber := 0;
   Program[7].Readings[1..4].MasterReadingNumber := 0;
   Program[8].Readings[1..4].MasterReadingNumber := 0;
   Program[1].Readings[1..4].LinkedMasterNumber := 0;
   Program[2].Readings[1..4].LinkedMasterNumber := 0;
   Program[3].Readings[1..4].LinkedMasterNumber := 0;
   Program[4].Readings[1..4].LinkedMasterNumber := 0;
   Program[5].Readings[1..4].LinkedMasterNumber := 0;
   Program[6].Readings[1..4].LinkedMasterNumber := 0;
   Program[7].Readings[1..4].LinkedMasterNumber := 0;
   Program[8].Readings[1..4].LinkedMasterNumber := 0;
   Program[1].Readings[1].Message[1..6].MessageType := 0;
   Program[1].Readings[2].Message[1..6].MessageType := 0;
   Program[1].Readings[3].Message[1..6].MessageType := 0;
   Program[1].Readings[4].Message[1..6].MessageType := 0;
   Program[2].Readings[1].Message[1..6].MessageType := 0;
   Program[2].Readings[2].Message[1..6].MessageType := 0;
   Program[2].Readings[3].Message[1..6].MessageType := 0;
   Program[2].Readings[4].Message[1..6].MessageType := 0;
   Program[3].Readings[1].Message[1..6].MessageType := 0;
   Program[3].Readings[2].Message[1..6].MessageType := 0;
   Program[3].Readings[3].Message[1..6].MessageType := 0;
   Program[3].Readings[4].Message[1..6].MessageType := 0;
   Program[4].Readings[1].Message[1..6].MessageType := 0;
   Program[4].Readings[2].Message[1..6].MessageType := 0;
   Program[4].Readings[3].Message[1..6].MessageType := 0;
   Program[4].Readings[4].Message[1..6].MessageType := 0;
   Program[5].Readings[1].Message[1..6].MessageType := 0;
   Program[5].Readings[2].Message[1..6].MessageType := 0;
   Program[5].Readings[3].Message[1..6].MessageType := 0;
   Program[5].Readings[4].Message[1..6].MessageType := 0;
   Program[6].Readings[1].Message[1..6].MessageType := 0;
   Program[6].Readings[2].Message[1..6].MessageType := 0;
   Program[6].Readings[3].Message[1..6].MessageType := 0;
   Program[6].Readings[4].Message[1..6].MessageType := 0;
   Program[7].Readings[1].Message[1..6].MessageType := 0;
   Program[7].Readings[2].Message[1..6].MessageType := 0;
   Program[7].Readings[3].Message[1..6].MessageType := 0;
   Program[7].Readings[4].Message[1..6].MessageType := 0;
   Program[8].Readings[1].Message[1..6].MessageType := 0;
   Program[8].Readings[2].Message[1..6].MessageType := 0;
   Program[8].Readings[3].Message[1..6].MessageType := 0;
   Program[8].Readings[4].Message[1..6].MessageType := 0;
   Program[1].Readings[1].Message[1..6].MessageFlagNumber := 0;
   Program[1].Readings[2].Message[1..6].MessageFlagNumber := 0;
   Program[1].Readings[3].Message[1..6].MessageFlagNumber := 0;
   Program[1].Readings[4].Message[1..6].MessageFlagNumber := 0;
   Program[2].Readings[1].Message[1..6].MessageFlagNumber := 0;
   Program[2].Readings[2].Message[1..6].MessageFlagNumber := 0;
   Program[2].Readings[3].Message[1..6].MessageFlagNumber := 0;
   Program[2].Readings[4].Message[1..6].MessageFlagNumber := 0;
   Program[3].Readings[1].Message[1..6].MessageFlagNumber := 0;
   Program[3].Readings[2].Message[1..6].MessageFlagNumber := 0;
   Program[3].Readings[3].Message[1..6].MessageFlagNumber := 0;
   Program[3].Readings[4].Message[1..6].MessageFlagNumber := 0;
   Program[4].Readings[1].Message[1..6].MessageFlagNumber := 0;
   Program[4].Readings[2].Message[1..6].MessageFlagNumber := 0;
   Program[4].Readings[3].Message[1..6].MessageFlagNumber := 0;
   Program[4].Readings[4].Message[1..6].MessageFlagNumber := 0;
   Program[5].Readings[1].Message[1..6].MessageFlagNumber := 0;
   Program[5].Readings[2].Message[1..6].MessageFlagNumber := 0;
   Program[5].Readings[3].Message[1..6].MessageFlagNumber := 0;
   Program[5].Readings[4].Message[1..6].MessageFlagNumber := 0;
   Program[6].Readings[1].Message[1..6].MessageFlagNumber := 0;
   Program[6].Readings[2].Message[1..6].MessageFlagNumber := 0;
   Program[6].Readings[3].Message[1..6].MessageFlagNumber := 0;
   Program[6].Readings[4].Message[1..6].MessageFlagNumber := 0;
   Program[7].Readings[1].Message[1..6].MessageFlagNumber := 0;
   Program[7].Readings[2].Message[1..6].MessageFlagNumber := 0;
   Program[7].Readings[3].Message[1..6].MessageFlagNumber := 0;
   Program[7].Readings[4].Message[1..6].MessageFlagNumber := 0;
   Program[8].Readings[1].Message[1..6].MessageFlagNumber := 0;
   Program[8].Readings[2].Message[1..6].MessageFlagNumber := 0;
   Program[8].Readings[3].Message[1..6].MessageFlagNumber := 0;
   Program[8].Readings[4].Message[1..6].MessageFlagNumber := 0;
END_DATA_BLOCK

DATA_BLOCK "safety_signals"   // DB2, F_DB
{ S7_Optimized_Access := 'TRUE' }
VERSION : 0.1
// stored: AutoNumber true, DBAccessibleFromOPCUA true, DBAccessibleFromWebserver true
   VAR
      estopok : Bool := FALSE;
      lightBarrierOk : Bool := FALSE;
      tableInPosition : Bool := FALSE;
      contactorsOk : Bool := FALSE;
      maintenanceDoorsClosed : Bool := FALSE;
      operateRobot1 : Bool := FALSE;
      serviceMode : Bool := FALSE;
      CoversClosed : Bool := FALSE;   // Emergency buttons and covers closed
      "3L+" : Bool := TRUE;   // emergency stop
      "4L+" : Bool := TRUE;   // emergency stop + service doors
      "5L+" : Bool := FALSE;   // emergency stop + service doors + light curtain
      serviceModeEnabled : Bool := FALSE;
      ACK_REI_Req : Bool := FALSE;
      RobotKeyNecessary : Bool := FALSE;
      Clock_1Hz : Bool := TRUE;
      doorUnlocked : Bool := FALSE;
   END_VAR
BEGIN
END_DATA_BLOCK

DATA_BLOCK "SandBoxData"   // DB22
{ S7_Optimized_Access := 'FALSE' }
VERSION : 0.1
// stored: AutoNumber false, DBAccessibleFromOPCUA true, DBAccessibleFromWebserver true, IsOnlyStoredInLoadMemory false, IsWriteProtectedInAS false
   VAR
      MnualCommandMem : Int := 6098;
      resetAuto : Bool := FALSE;
      rivetingStartedMem : Bool;
   END_VAR
BEGIN
END_DATA_BLOCK

DATA_BLOCK "AnalogData"   // DB27
{ S7_Optimized_Access := 'FALSE' }
VERSION : 0.1
// stored: AutoNumber false, DBAccessibleFromOPCUA true, DBAccessibleFromWebserver true, IsOnlyStoredInLoadMemory false, IsWriteProtectedInAS false
   VAR
      InputResults : Array[1..12] of Real;
      OutputsRequired : Array[1..8] of Real;
      OutputsRequiredHMI : Array[1..8] of Int;
   END_VAR
BEGIN
   InputResults[1] := 7.960068;
   InputResults[2] := 8.440392;
   InputResults[3] := 7.105035;
   InputResults[4] := 7.011719;
   InputResults[5..12] := 0.0;
   OutputsRequired[1..8] := 0.0;
   OutputsRequiredHMI[1..8] := 16#0000;
END_DATA_BLOCK

DATA_BLOCK "CylindersHMI"   // DB50
{ S7_Optimized_Access := 'TRUE' }
VERSION : 0.1
// stored: AutoNumber true, DBAccessibleFromOPCUA true, DBAccessibleFromWebserver true, IsOnlyStoredInLoadMemory false, IsRetainMemResEnabled false, IsWriteProtectedInAS false, MemoryReserve 100
   VAR
      Status : Array[0.."NumberOfCylinders"] of Int;
      SelectedCylinderCylinderCommand : Int := 0;
      SelectedCylinder : Int := 0;
      SelectedCylinderStatus : Int := 0;
      SelectedCylinder_1 : Int := 0;
      SelectedCylinder_2 : Int := 0;
      SelectedCylinder_3 : Int := 0;
      SelectedCylinder_4 : Int := 0;
      SelectedCylinderStatus_1 : Int := 0;
      SelectedCylinderStatus_2 : Int := 0;
      SelectedCylinderStatus_3 : Int := 0;
      SelectedCylinderStatus_4 : Int := 0;
      DisableHMIControl : Bool := FALSE;
      CylinderInfoHMI : Int := -1;
      CylinderInfoHMIAction : Int := 0;
   END_VAR
BEGIN
   Status[0..4] := 257;
   Status[5..6] := 1;
   Status[7..8] := 257;
   Status[9..10] := 1;
   Status[11..14] := 257;
   Status[15..16] := 1;
   Status[17] := 2;
   Status[18] := 1;
   Status[19] := 0;
END_DATA_BLOCK

DATA_BLOCK "DiagnosticConfigured"   // DB38
{ S7_Optimized_Access := 'TRUE' }
VERSION : 0.1
// stored: AutoNumber true, DBAccessibleFromOPCUA true, DBAccessibleFromWebserver true, IsOnlyStoredInLoadMemory false, IsRetainMemResEnabled false, IsWriteProtectedInAS false, MemoryReserve 100
   VAR
      Adresses : Array[1..255] of Int;
      Errors : Array[1..255] of Bool;
      Exists : Array[1..255] of Bool;
      States : Array[1..255] of Int;
      Updated : Bool := FALSE;
   END_VAR
BEGIN
   Adresses[1] := 11;
   Adresses[2] := 31;
   Adresses[3] := 32;
   Adresses[4] := 33;
   Adresses[5] := 34;
   Adresses[6] := 41;
   Adresses[7] := 61;
   Adresses[8] := 62;
   Adresses[9] := 63;
   Adresses[10] := 64;
   Adresses[11] := 65;
   Adresses[12] := 66;
   Adresses[13] := 68;
   Adresses[14] := 69;
   Adresses[15] := 70;
   Adresses[16] := 71;
   Adresses[17] := 73;
   Adresses[18] := 74;
   Adresses[19] := 91;
   Adresses[20..255] := 0;
   Errors[1..255] := FALSE;
   Exists[1..19] := TRUE;
   Exists[20..255] := FALSE;
   States[1..19] := 1;
   States[20..255] := 0;
END_DATA_BLOCK

DATA_BLOCK "HydraulicManualMode"   // DB14
{ S7_Optimized_Access := 'TRUE' }
VERSION : 0.1
// stored: AutoNumber true, DBAccessibleFromOPCUA true, DBAccessibleFromWebserver true, IsOnlyStoredInLoadMemory false, IsRetainMemResEnabled false, IsWriteProtectedInAS false, MemoryReserve 100
   VAR
      RivetingCylinderActiveHMI : Bool;
      CupformingCylinderActiveHMI : Bool;
   END_VAR
BEGIN
END_DATA_BLOCK

DATA_BLOCK "PartHolderData"   // DB21
{ S7_Optimized_Access := 'TRUE' }
VERSION : 0.1
// stored: AutoNumber true, DBAccessibleFromOPCUA true, DBAccessibleFromWebserver true, IsOnlyStoredInLoadMemory false, IsRetainMemResEnabled false, IsWriteProtectedInAS false, MemoryReserve 100
   VAR RETAIN
      OkUpperStockAmountSideA : USInt := 1;
      OkLowerStockAmountSideA : USInt := 0;
      NOKBoxAmount : USInt := 1;
   END_VAR
   VAR
      NOKBoxFull : Bool := FALSE;
      ConfirmEmptyOKStock : Bool := FALSE;
      ConfirmEmptyNOKBox : Bool := FALSE;
      EmptyOKStockConfirmed : Bool := FALSE;
      EmptyNOKBoxConfirmed : Bool := FALSE;
      NOKBoxActivated : Bool := FALSE;
      NOKBoxPesent : Bool := TRUE;
      OKholderPresent : Bool := TRUE;
      OKholderReadySideA : Bool := FALSE;
      OKholderReadySideB : Bool;
   END_VAR
   VAR RETAIN
      OkUpperStockAmountSideB : USInt := 0;
      OkLowerStockAmountSideB : USInt := 0;
   END_VAR
BEGIN
END_DATA_BLOCK

DATA_BLOCK "DB_STATUS_IJCORE"   // DB69
{ S7_Optimized_Access := 'TRUE' }
VERSION : 0.1
// stored: AutoNumber true, DBAccessibleFromOPCUA true, DBAccessibleFromWebserver true, IsOnlyStoredInLoadMemory false, IsRetainMemResEnabled false, IsWriteProtectedInAS false, MemoryReserve 100
   VAR
      CONFIG_MSG { S7_SetPoint := 'True'} : Array[0..30] of "CONFIG_MSG_IJC";
      EDIT_MSG { S7_SetPoint := 'True'} : "CONFIG_MSG_IJC";
      INDEX_EDITADO { S7_SetPoint := 'True'} : Int := 1;
      INDEX_EDITADO_ANTERIOR : Int := 1;
      PB_VALIDAR_EDICION { S7_SetPoint := 'True'} : Bool := FALSE;
      ANSWER_RECIB : Array[0..30] of Int;
      ANSWER_NFP : Array[0..5] of Int;
      ANSWER_TRB : Array[0..5] of Int;
      ANSWER_STA : Array[0..5] of Int;
      ANSWER_TRC : Array[0..5] of Int;
      ANSWER_TRW : Array[0..5] of Int;
      ANSWER_TRI : Array[0..5] of Int;
      DN_TRC_COMP : Array[0..5] of Bool;
      ALL_TRC_OK : Bool;
      ALL_CNF_OK : Bool;
      ALL_TRR_OK : Bool;
      INDEX_ENVIO : DInt := 40;
      INDEX_MSG_CONFIG : DInt;
      ALARMA : Array[0..10] of Word;
      INDEX_ANSWER_STA : Int := 0;
      INDEX_ANSWER_TRC : Int := 9;
      INDEX_ANSWER_TRW : Int := 15;
      INDEX_ANSWER_TRI : Int := 10;
      INDEX_CLEAR : Int;
      INDEX_HMI : Int;
      PAGINA_HMI : Int;
      PAGINA_UP : Bool;
      PAGINA_DOWN : Bool;
      HMI_M_TYPE : Array[0..10] of String;
      HMI_M_NBR : Array[0..10] of DInt;
      HMI_ANS : Array[0..10] of SInt;
      HMI_STEP : Array[0..10] of Int;
      HMI_FLT : Array[0..10] of Bool;
      HMI_DN : Array[0..10] of Bool;
      HMI : Array[0..10] of Struct
         SEND : Struct
            MSG : String[50];
            SW : SInt;
         END_STRUCT;
         RCV : Struct
            MSG : String[50];
            SW : SInt;
         END_STRUCT;
      END_STRUCT;
      AW_number : DInt;
      AW_duration : Time;
      AW_durationMax : Time;
      Restart_Counter_bit_of_life : Int;
      AW_duration_fault : Time;
      R_NBR_MESSAGE : DInt;
      MES_DIAG_MESSAGE_NBR : Int := 1;
      S_DURATION_FAULT : Int := 30;
      R_DURATION_FAULT : Int := 30;
      S_DURATION : Int;
      S_MAX_DURATION : Int;
      S_NBR_MESSAGE : DInt;
      R_DURATION : Int;
      R_MAX_DURATION : Int;
      MES_RESET_AW_DIAG : Bool;
      MES_RESET_MESS_DIAG : Bool;
      MES_TEMP_S_FT : Int := 30;
      MES_TEMP_R_FT : Int := 30;
      MES_TEMP_NBR_MESS : Int := 1;
   END_VAR
BEGIN
   CONFIG_MSG[1..4]."TYPE" := 'STA';
   CONFIG_MSG[5..8]."TYPE" := 'TRC';
   CONFIG_MSG[9..10]."TYPE" := 'TRR';
   CONFIG_MSG[11..14]."TYPE" := 'CNF';
   CONFIG_MSG[15]."TYPE" := 'PFC';
   EDIT_MSG."TYPE" := '';
   EDIT_MSG.KANBAN := '';
   EDIT_MSG.COMPONENT := '';
   EDIT_MSG.START := FALSE;
   EDIT_MSG.PROCESS_STATUS := 0;
   ANSWER_RECIB[0..2] := 0;
   ANSWER_RECIB[3] := 1;
   ANSWER_RECIB[4..5] := 8224;
   ANSWER_RECIB[6] := 1;
   ANSWER_RECIB[7..8] := 8224;
   ANSWER_RECIB[9..11] := 0;
   ANSWER_RECIB[12] := 1;
   ANSWER_RECIB[13..14] := 8224;
   ANSWER_RECIB[15..18] := 0;
   ANSWER_RECIB[19] := 1;
   ANSWER_RECIB[20] := 8224;
   ANSWER_NFP[0..2] := 0;
   ANSWER_NFP[3] := 1;
   ANSWER_NFP[4..5] := 8224;
   ANSWER_TRB[0..5] := 0;
   ANSWER_STA[0..2] := 0;
   ANSWER_STA[3..4] := 1;
   ANSWER_STA[5] := 0;
   ANSWER_TRC[0..5] := 0;
   ANSWER_TRW[0..5] := 0;
   ANSWER_TRI[0..5] := 0;
   DN_TRC_COMP[0..5] := FALSE;
   ALARMA[0..10] := 16#0000;
END_DATA_BLOCK

DATA_BLOCK "PartErrorsCounter"   // DB46
{ S7_Optimized_Access := 'TRUE' }
VERSION : 0.1
// stored: AutoNumber true, DBAccessibleFromOPCUA true, DBAccessibleFromWebserver true, IsOnlyStoredInLoadMemory false, IsRetainMemResEnabled false, IsWriteProtectedInAS false, MemoryReserve 100
   VAR RETAIN
      CountersRef { S7_SetPoint := 'True'} : Array[1.."NumberOfProductionPrograms"] of "UDT_NOKcounter";
   END_VAR
   VAR
      CountersHMI : "UDT_NOKcounter";
   END_VAR
BEGIN
   CountersRef[1].Counters[0,0..50] := 0;
   CountersRef[1].Counters[1,0..9] := 0;
   CountersRef[1].Counters[1,10] := 2;
   CountersRef[1].Counters[1,11] := 1;
   CountersRef[1].Counters[1,12..19] := 0;
   CountersRef[1].Counters[1,20] := 3;
   CountersRef[1].Counters[1,21] := 1;
   CountersRef[1].Counters[1,22..33] := 0;
   CountersRef[1].Counters[1,34] := 1;
   CountersRef[1].Counters[1,35..43] := 0;
   CountersRef[1].Counters[1,44] := 1;
   CountersRef[1].Counters[1,45..50] := 0;
   CountersRef[1].Counters[2,0..13] := 0;
   CountersRef[1].Counters[2,14] := 1;
   CountersRef[1].Counters[2,15..20] := 0;
   CountersRef[1].Counters[2,21] := 1;
   CountersRef[1].Counters[2,22..50] := 0;
   CountersRef[1].Counters[3,0..50] := 0;
   CountersRef[2].Counters[0,0..50] := 0;
   CountersRef[2].Counters[1,0..9] := 0;
   CountersRef[2].Counters[1,10] := 4;
   CountersRef[2].Counters[1,11] := 1;
   CountersRef[2].Counters[1,12..19] := 0;
   CountersRef[2].Counters[1,20] := 3;
   CountersRef[2].Counters[1,21] := 2;
   CountersRef[2].Counters[1,22..50] := 0;
   CountersRef[2].Counters[2,0..10] := 0;
   CountersRef[2].Counters[2,11] := 1;
   CountersRef[2].Counters[2,12..13] := 0;
   CountersRef[2].Counters[2,14] := 1;
   CountersRef[2].Counters[2,15..20] := 0;
   CountersRef[2].Counters[2,21] := 1;
   CountersRef[2].Counters[2,22..23] := 0;
   CountersRef[2].Counters[2,24] := 1;
   CountersRef[2].Counters[2,25..30] := 0;
   CountersRef[2].Counters[2,31] := 1;
   CountersRef[2].Counters[2,32..33] := 0;
   CountersRef[2].Counters[2,34] := 1;
   CountersRef[2].Counters[2,35..40] := 0;
   CountersRef[2].Counters[2,41] := 1;
   CountersRef[2].Counters[2,42..43] := 0;
   CountersRef[2].Counters[2,44] := 1;
   CountersRef[2].Counters[2,45..50] := 0;
   CountersRef[2].Counters[3,0..50] := 0;
   CountersRef[3].Counters[0,0..50] := 0;
   CountersRef[3].Counters[1,0..50] := 0;
   CountersRef[3].Counters[2,0..50] := 0;
   CountersRef[3].Counters[3,0..50] := 0;
   CountersRef[4].Counters[0,0..50] := 0;
   CountersRef[4].Counters[1,0..50] := 0;
   CountersRef[4].Counters[2,0..50] := 0;
   CountersRef[4].Counters[3,0..50] := 0;
   CountersRef[5].Counters[0,0..50] := 0;
   CountersRef[5].Counters[1,0..9] := 0;
   CountersRef[5].Counters[1,10] := 17;
   CountersRef[5].Counters[1,11] := 6;
   CountersRef[5].Counters[1,12..19] := 0;
   CountersRef[5].Counters[1,20..21] := 1;
   CountersRef[5].Counters[1,22..50] := 0;
   CountersRef[5].Counters[2,0..9] := 0;
   CountersRef[5].Counters[2,10] := 4;
   CountersRef[5].Counters[2,11] := 3;
   CountersRef[5].Counters[2,12..13] := 0;
   CountersRef[5].Counters[2,14] := 1;
   CountersRef[5].Counters[2,15..23] := 0;
   CountersRef[5].Counters[2,24] := 4;
   CountersRef[5].Counters[2,25..50] := 0;
   CountersRef[5].Counters[3,0..50] := 0;
   CountersRef[6].Counters[0,0..50] := 0;
   CountersRef[6].Counters[1,0..50] := 0;
   CountersRef[6].Counters[2,0..9] := 0;
   CountersRef[6].Counters[2,10] := 1;
   CountersRef[6].Counters[2,11..13] := 0;
   CountersRef[6].Counters[2,14] := 1;
   CountersRef[6].Counters[2,15..21] := 0;
   CountersRef[6].Counters[2,22] := 1;
   CountersRef[6].Counters[2,23..33] := 0;
   CountersRef[6].Counters[2,34] := 2;
   CountersRef[6].Counters[2,35..43] := 0;
   CountersRef[6].Counters[2,44] := 2;
   CountersRef[6].Counters[2,45..50] := 0;
   CountersRef[6].Counters[3,0..50] := 0;
   CountersRef[7].Counters[0,0..50] := 0;
   CountersRef[7].Counters[1,0..50] := 0;
   CountersRef[7].Counters[2,0..50] := 0;
   CountersRef[7].Counters[3,0..50] := 0;
   CountersRef[8].Counters[0,0..50] := 0;
   CountersRef[8].Counters[1,0..50] := 0;
   CountersRef[8].Counters[2,0..50] := 0;
   CountersRef[8].Counters[3,0..50] := 0;
   CountersHMI.Counters[0,0..50] := 0;
   CountersHMI.Counters[1,0..50] := 0;
   CountersHMI.Counters[2,0..50] := 0;
   CountersHMI.Counters[3,0..50] := 0;
END_DATA_BLOCK

DATA_BLOCK "READER_MODEL"   // DB74
{ S7_Optimized_Access := 'TRUE' }
VERSION : 0.1
// stored: AutoNumber true, DBAccessibleFromOPCUA true, DBAccessibleFromWebserver true, IsOnlyStoredInLoadMemory false, IsRetainMemResEnabled false, IsWriteProtectedInAS false, MemoryReserve 100
   VAR RETAIN
      PRODUCT { S7_SetPoint := 'True'} : Array[0.."NumberOfProductionPrograms"] of "READER_PRODUCT";
   END_VAR
BEGIN
   PRODUCT[1..4].SIDE_RH.POSITION := 13;
   PRODUCT[1..4].SIDE_RH.LEN := 3;
   PRODUCT[1].SIDE_RH.STRING_LABEL := '336';
   PRODUCT[2].SIDE_RH.STRING_LABEL := '532';
   PRODUCT[3].SIDE_RH.STRING_LABEL := '336';
   PRODUCT[4].SIDE_RH.STRING_LABEL := '532';
   PRODUCT[1..4].SIDE_RH.READER_BYPASS := FALSE;
   PRODUCT[1..4].SIDE_LH.POSITION := 13;
   PRODUCT[1..4].SIDE_LH.LEN := 3;
   PRODUCT[1].SIDE_LH.STRING_LABEL := '328';
   PRODUCT[2].SIDE_LH.STRING_LABEL := '526';
   PRODUCT[3].SIDE_LH.STRING_LABEL := '328';
   PRODUCT[4].SIDE_LH.STRING_LABEL := '526';
   PRODUCT[1..4].SIDE_LH.READER_BYPASS := FALSE;
   PRODUCT[1..4].REAR_TUBE.POSITION := 13;
   PRODUCT[1..4].REAR_TUBE.LEN := 3;
   PRODUCT[1].REAR_TUBE.STRING_LABEL := '343';
   PRODUCT[2].REAR_TUBE.STRING_LABEL := '514';
   PRODUCT[3].REAR_TUBE.STRING_LABEL := '343';
   PRODUCT[4].REAR_TUBE.STRING_LABEL := '514';
   PRODUCT[1..4].REAR_TUBE.READER_BYPASS := FALSE;
   PRODUCT[1..2].FRONT_TUBE.POSITION := 13;
   PRODUCT[1..2].FRONT_TUBE.LEN := 3;
   PRODUCT[1..2].FRONT_TUBE.STRING_LABEL := '907';
   PRODUCT[1].FRONT_TUBE.READER_BYPASS := FALSE;
   PRODUCT[2..4].FRONT_TUBE.READER_BYPASS := TRUE;
   PRODUCT[1..2].NUM_TUBE := TRUE;
   PRODUCT[3].NUM_TUBE := FALSE;
END_DATA_BLOCK

